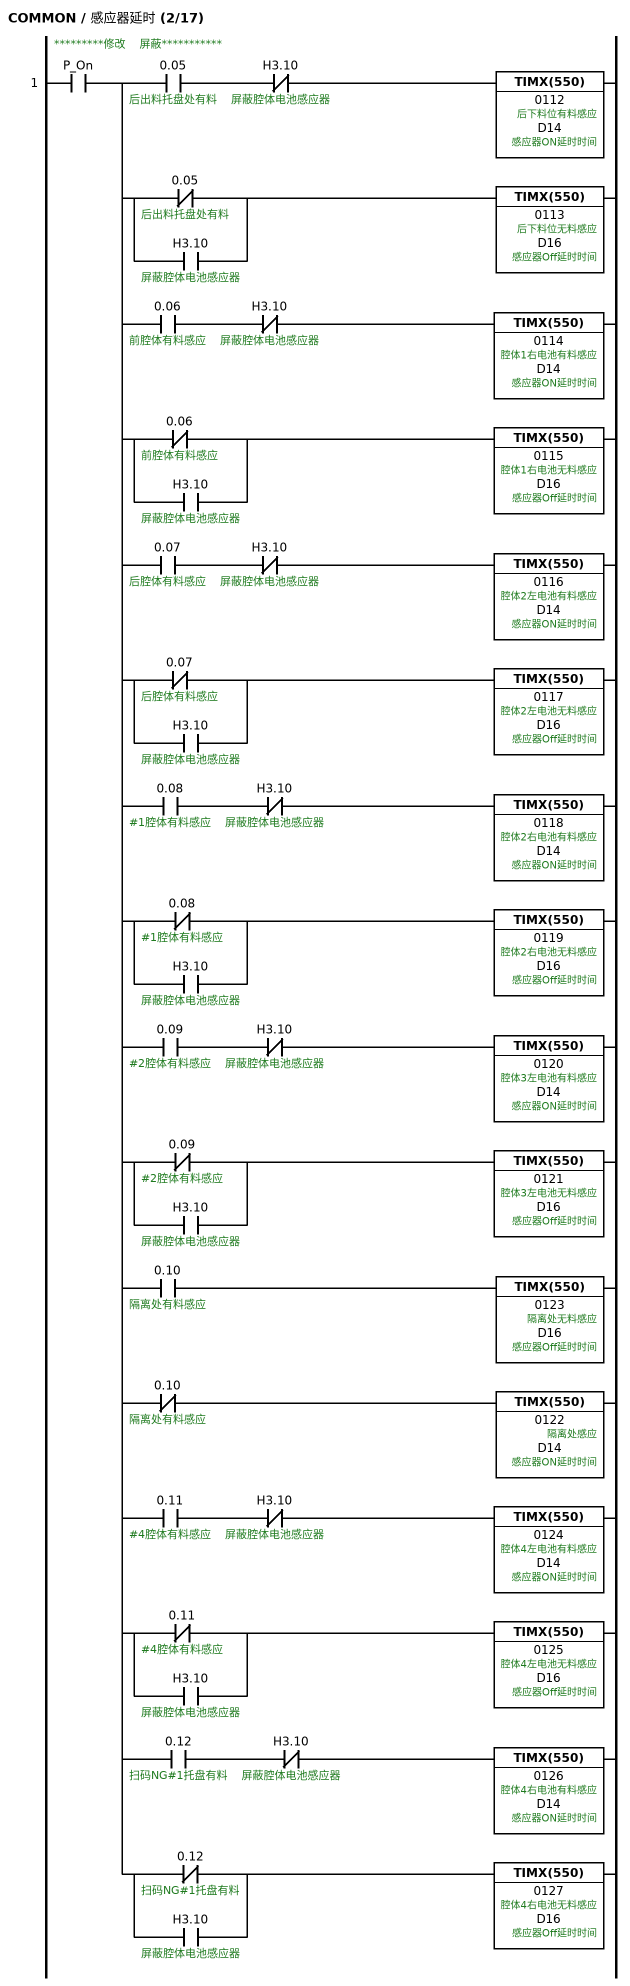
; [picture p408: COMMON / 感应器延时, rungs 1-1]
; rung 1: *********修改    屏蔽***********
LD P_On
OUT TR0
AND 0.05  ; 后出料托盘处有料
ANDNOT H3.10  ; 屏蔽腔体电池感应器
TIMX(550) 0112 D14  ; 感应器ON延时时间, 后下料位有料感应
LD TR0
LDNOT 0.05  ; 后出料托盘处有料
OR H3.10  ; 屏蔽腔体电池感应器
ANDLD
TIMX(550) 0113 D16  ; 感应器Off延时时间, 后下料位无料感应
LD TR0
AND 0.06  ; 前腔体有料感应
ANDNOT H3.10  ; 屏蔽腔体电池感应器
TIMX(550) 0114 D14  ; 感应器ON延时时间, 腔体1右电池有料感应
LD TR0
LDNOT 0.06  ; 前腔体有料感应
OR H3.10  ; 屏蔽腔体电池感应器
ANDLD
TIMX(550) 0115 D16  ; 感应器Off延时时间, 腔体1右电池无料感应
LD TR0
AND 0.07  ; 后腔体有料感应
ANDNOT H3.10  ; 屏蔽腔体电池感应器
TIMX(550) 0116 D14  ; 感应器ON延时时间, 腔体2左电池有料感应
LD TR0
LDNOT 0.07  ; 后腔体有料感应
OR H3.10  ; 屏蔽腔体电池感应器
ANDLD
TIMX(550) 0117 D16  ; 感应器Off延时时间, 腔体2左电池无料感应
LD TR0
AND 0.08  ; #1腔体有料感应
ANDNOT H3.10  ; 屏蔽腔体电池感应器
TIMX(550) 0118 D14  ; 感应器ON延时时间, 腔体2右电池有料感应
LD TR0
LDNOT 0.08  ; #1腔体有料感应
OR H3.10  ; 屏蔽腔体电池感应器
ANDLD
TIMX(550) 0119 D16  ; 感应器Off延时时间, 腔体2右电池无料感应
LD TR0
AND 0.09  ; #2腔体有料感应
ANDNOT H3.10  ; 屏蔽腔体电池感应器
TIMX(550) 0120 D14  ; 感应器ON延时时间, 腔体3左电池有料感应
LD TR0
LDNOT 0.09  ; #2腔体有料感应
OR H3.10  ; 屏蔽腔体电池感应器
ANDLD
TIMX(550) 0121 D16  ; 感应器Off延时时间, 腔体3左电池无料感应
LD TR0
AND 0.10  ; 隔离处有料感应
TIMX(550) 0123 D16  ; 感应器Off延时时间, 隔离处无料感应
LD TR0
ANDNOT 0.10  ; 隔离处有料感应
TIMX(550) 0122 D14  ; 感应器ON延时时间, 隔离处感应
LD TR0
AND 0.11  ; #4腔体有料感应
ANDNOT H3.10  ; 屏蔽腔体电池感应器
TIMX(550) 0124 D14  ; 感应器ON延时时间, 腔体4左电池有料感应
LD TR0
LDNOT 0.11  ; #4腔体有料感应
OR H3.10  ; 屏蔽腔体电池感应器
ANDLD
TIMX(550) 0125 D16  ; 感应器Off延时时间, 腔体4左电池无料感应
LD TR0
AND 0.12  ; 扫码NG#1托盘有料
ANDNOT H3.10  ; 屏蔽腔体电池感应器
TIMX(550) 0126 D14  ; 感应器ON延时时间, 腔体4右电池有料感应
LD TR0
LDNOT 0.12  ; 扫码NG#1托盘有料
OR H3.10  ; 屏蔽腔体电池感应器
ANDLD
TIMX(550) 0127 D16  ; 感应器Off延时时间, 腔体4右电池无料感应

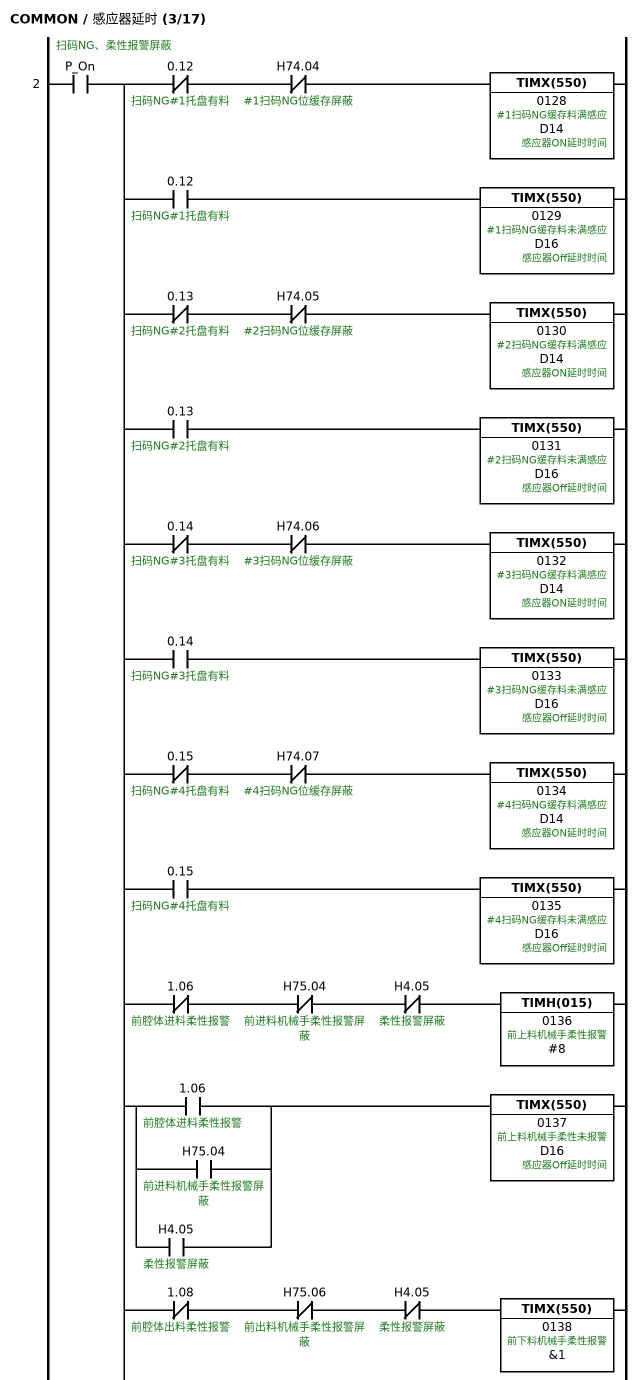

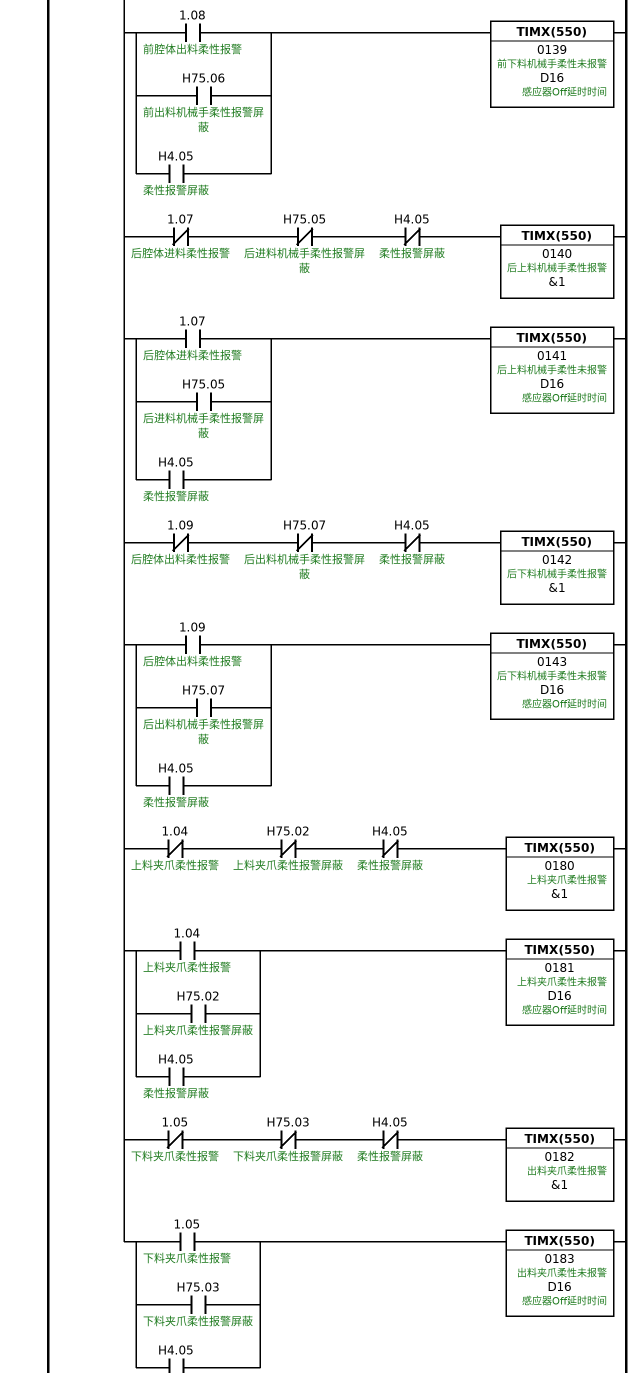

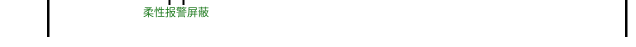
; rung 2: 扫码NG、柔性报警屏蔽
LD P_On
OUT TR0
ANDNOT 0.12  ; 扫码NG#1托盘有料
ANDNOT H74.04  ; #1扫码NG位缓存屏蔽
TIMX(550) 0128 D14  ; 感应器ON延时时间, #1扫码NG缓存料满感应
LD TR0
AND 0.12  ; 扫码NG#1托盘有料
TIMX(550) 0129 D16  ; 感应器Off延时时间, #1扫码NG缓存料未满感应
LD TR0
ANDNOT 0.13  ; 扫码NG#2托盘有料
ANDNOT H74.05  ; #2扫码NG位缓存屏蔽
TIMX(550) 0130 D14  ; 感应器ON延时时间, #2扫码NG缓存料满感应
LD TR0
AND 0.13  ; 扫码NG#2托盘有料
TIMX(550) 0131 D16  ; 感应器Off延时时间, #2扫码NG缓存料未满感应
LD TR0
ANDNOT 0.14  ; 扫码NG#3托盘有料
ANDNOT H74.06  ; #3扫码NG位缓存屏蔽
TIMX(550) 0132 D14  ; 感应器ON延时时间, #3扫码NG缓存料满感应
LD TR0
AND 0.14  ; 扫码NG#3托盘有料
TIMX(550) 0133 D16  ; 感应器Off延时时间, #3扫码NG缓存料未满感应
LD TR0
ANDNOT 0.15  ; 扫码NG#4托盘有料
ANDNOT H74.07  ; #4扫码NG位缓存屏蔽
TIMX(550) 0134 D14  ; 感应器ON延时时间, #4扫码NG缓存料满感应
LD TR0
AND 0.15  ; 扫码NG#4托盘有料
TIMX(550) 0135 D16  ; 感应器Off延时时间, #4扫码NG缓存料未满感应
LD TR0
ANDNOT 1.06  ; 前腔体进料柔性报警
ANDNOT H75.04  ; 前进料机械手柔性报警屏蔽
ANDNOT H4.05  ; 柔性报警屏蔽
TIMH(015) 0136 #8  ; 前上料机械手柔性报警
LD TR0
LD 1.06  ; 前腔体进料柔性报警
OR H75.04  ; 前进料机械手柔性报警屏蔽
OR H4.05  ; 柔性报警屏蔽
ANDLD
TIMX(550) 0137 D16  ; 感应器Off延时时间, 前上料机械手柔性未报警
LD TR0
ANDNOT 1.08  ; 前腔体出料柔性报警
ANDNOT H75.06  ; 前出料机械手柔性报警屏蔽
ANDNOT H4.05  ; 柔性报警屏蔽
TIMX(550) 0138 &1  ; 前下料机械手柔性报警
LD TR0
LD 1.08  ; 前腔体出料柔性报警
OR H75.06  ; 前出料机械手柔性报警屏蔽
OR H4.05  ; 柔性报警屏蔽
ANDLD
TIMX(550) 0139 D16  ; 感应器Off延时时间, 前下料机械手柔性未报警
LD TR0
ANDNOT 1.07  ; 后腔体进料柔性报警
ANDNOT H75.05  ; 后进料机械手柔性报警屏蔽
ANDNOT H4.05  ; 柔性报警屏蔽
TIMX(550) 0140 &1  ; 后上料机械手柔性报警
LD TR0
LD 1.07  ; 后腔体进料柔性报警
OR H75.05  ; 后进料机械手柔性报警屏蔽
OR H4.05  ; 柔性报警屏蔽
ANDLD
TIMX(550) 0141 D16  ; 感应器Off延时时间, 后上料机械手柔性未报警
LD TR0
ANDNOT 1.09  ; 后腔体出料柔性报警
ANDNOT H75.07  ; 后出料机械手柔性报警屏蔽
ANDNOT H4.05  ; 柔性报警屏蔽
TIMX(550) 0142 &1  ; 后下料机械手柔性报警
LD TR0
LD 1.09  ; 后腔体出料柔性报警
OR H75.07  ; 后出料机械手柔性报警屏蔽
OR H4.05  ; 柔性报警屏蔽
ANDLD
TIMX(550) 0143 D16  ; 感应器Off延时时间, 后下料机械手柔性未报警
LD TR0
ANDNOT 1.04  ; 上料夹爪柔性报警
ANDNOT H75.02  ; 上料夹爪柔性报警屏蔽
ANDNOT H4.05  ; 柔性报警屏蔽
TIMX(550) 0180 &1  ; 上料夹爪柔性报警
LD TR0
LD 1.04  ; 上料夹爪柔性报警
OR H75.02  ; 上料夹爪柔性报警屏蔽
OR H4.05  ; 柔性报警屏蔽
ANDLD
TIMX(550) 0181 D16  ; 感应器Off延时时间, 上料夹爪柔性未报警
LD TR0
ANDNOT 1.05  ; 下料夹爪柔性报警
ANDNOT H75.03  ; 下料夹爪柔性报警屏蔽
ANDNOT H4.05  ; 柔性报警屏蔽
TIMX(550) 0182 &1  ; 出料夹爪柔性报警
LD TR0
LD 1.05  ; 下料夹爪柔性报警
OR H75.03  ; 下料夹爪柔性报警屏蔽
OR H4.05  ; 柔性报警屏蔽
ANDLD
TIMX(550) 0183 D16  ; 感应器Off延时时间, 出料夹爪柔性未报警

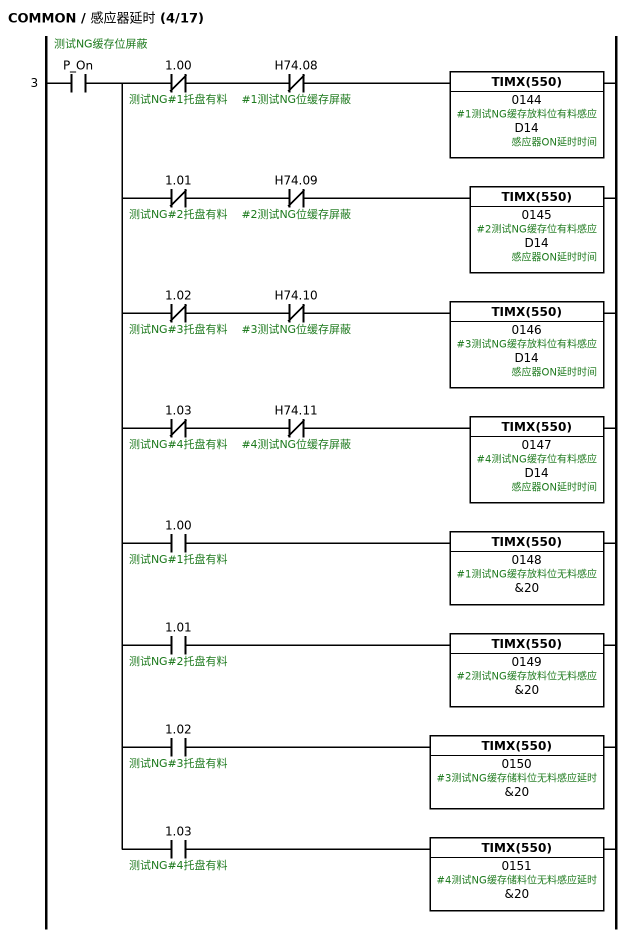
; rung 3: 测试NG缓存位屏蔽
LD P_On
OUT TR0
ANDNOT 1.00  ; 测试NG#1托盘有料
ANDNOT H74.08  ; #1测试NG位缓存屏蔽
TIMX(550) 0144 D14  ; 感应器ON延时时间, #1测试NG缓存放料位有料感应
LD TR0
ANDNOT 1.01  ; 测试NG#2托盘有料
ANDNOT H74.09  ; #2测试NG位缓存屏蔽
TIMX(550) 0145 D14  ; 感应器ON延时时间, #2测试NG缓存位有料感应
LD TR0
ANDNOT 1.02  ; 测试NG#3托盘有料
ANDNOT H74.10  ; #3测试NG位缓存屏蔽
TIMX(550) 0146 D14  ; 感应器ON延时时间, #3测试NG缓存放料位有料感应
LD TR0
ANDNOT 1.03  ; 测试NG#4托盘有料
ANDNOT H74.11  ; #4测试NG位缓存屏蔽
TIMX(550) 0147 D14  ; 感应器ON延时时间, #4测试NG缓存位有料感应
LD TR0
AND 1.00  ; 测试NG#1托盘有料
TIMX(550) 0148 &20  ; #1测试NG缓存放料位无料感应
LD TR0
AND 1.01  ; 测试NG#2托盘有料
TIMX(550) 0149 &20  ; #2测试NG缓存放料位无料感应
LD TR0
AND 1.02  ; 测试NG#3托盘有料
TIMX(550) 0150 &20  ; #3测试NG缓存储料位无料感应延时
LD TR0
AND 1.03  ; 测试NG#4托盘有料
TIMX(550) 0151 &20  ; #4测试NG缓存储料位无料感应延时

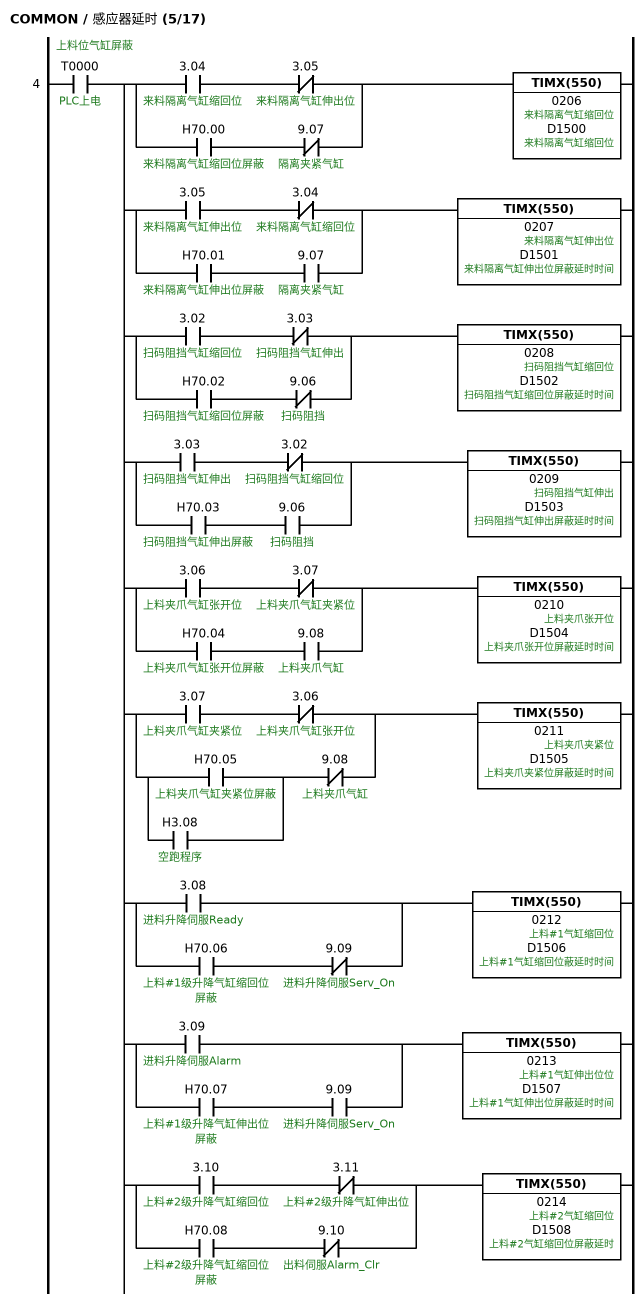

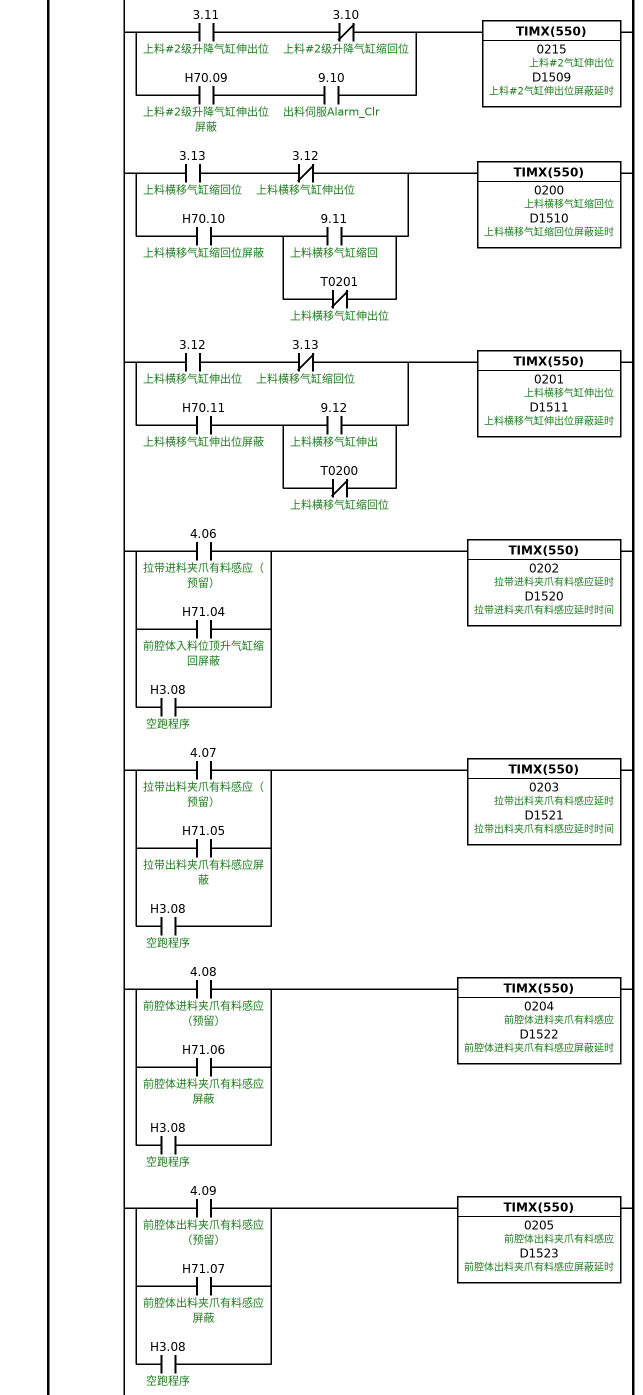

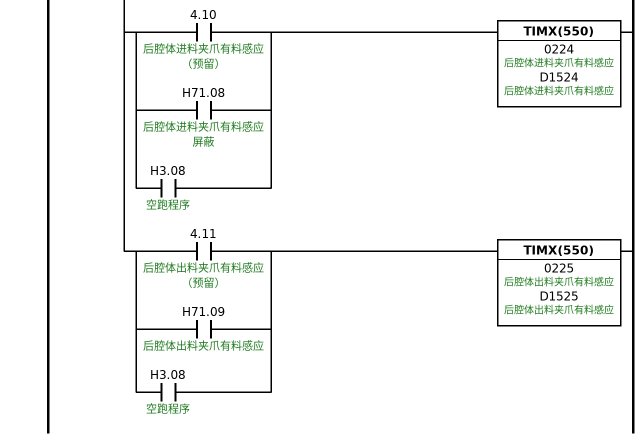
; rung 4: 上料位气缸屏蔽
LD T0000  ; PLC上电
OUT TR0
LD 3.04  ; 来料隔离气缸缩回位
ANDNOT 3.05  ; 来料隔离气缸伸出位
LD H70.00  ; 来料隔离气缸缩回位屏蔽
ANDNOT 9.07  ; 隔离夹紧气缸
ORLD
ANDLD
TIMX(550) 0206 D1500  ; 来料隔离气缸缩回位
LD TR0
LD 3.05  ; 来料隔离气缸伸出位
ANDNOT 3.04  ; 来料隔离气缸缩回位
LD H70.01  ; 来料隔离气缸伸出位屏蔽
AND 9.07  ; 隔离夹紧气缸
ORLD
ANDLD
TIMX(550) 0207 D1501  ; 来料隔离气缸伸出位屏蔽延时时间, 来料隔离气缸伸出位
LD TR0
LD 3.02  ; 扫码阻挡气缸缩回位
ANDNOT 3.03  ; 扫码阻挡气缸伸出
LD H70.02  ; 扫码阻挡气缸缩回位屏蔽
ANDNOT 9.06  ; 扫码阻挡
ORLD
ANDLD
TIMX(550) 0208 D1502  ; 扫码阻挡气缸缩回位屏蔽延时时间, 扫码阻挡气缸缩回位
LD TR0
LD 3.03  ; 扫码阻挡气缸伸出
ANDNOT 3.02  ; 扫码阻挡气缸缩回位
LD H70.03  ; 扫码阻挡气缸伸出屏蔽
AND 9.06  ; 扫码阻挡
ORLD
ANDLD
TIMX(550) 0209 D1503  ; 扫码阻挡气缸伸出屏蔽延时时间, 扫码阻挡气缸伸出
LD TR0
LD 3.06  ; 上料夹爪气缸张开位
ANDNOT 3.07  ; 上料夹爪气缸夹紧位
LD H70.04  ; 上料夹爪气缸张开位屏蔽
AND 9.08  ; 上料夹爪气缸
ORLD
ANDLD
TIMX(550) 0210 D1504  ; 上料夹爪张开位屏蔽延时时间, 上料夹爪张开位
LD TR0
LD 3.07  ; 上料夹爪气缸夹紧位
ANDNOT 3.06  ; 上料夹爪气缸张开位
LD H70.05  ; 上料夹爪气缸夹紧位屏蔽
OR H3.08  ; 空跑程序
ANDNOT 9.08  ; 上料夹爪气缸
ORLD
ANDLD
TIMX(550) 0211 D1505  ; 上料夹爪夹紧位屏蔽延时时间, 上料夹爪夹紧位
LD TR0
LD 3.08  ; 进料升降伺服Ready
LD H70.06  ; 上料#1级升降气缸缩回位屏蔽
ANDNOT 9.09  ; 进料升降伺服Serv_On
ORLD
ANDLD
TIMX(550) 0212 D1506  ; 上料#1气缸缩回位蔽延时时间, 上料#1气缸缩回位
LD TR0
LD 3.09  ; 进料升降伺服Alarm
LD H70.07  ; 上料#1级升降气缸伸出位屏蔽
AND 9.09  ; 进料升降伺服Serv_On
ORLD
ANDLD
TIMX(550) 0213 D1507  ; 上料#1气缸伸出位屏蔽延时时间, 上料#1气缸伸出位位
LD TR0
LD 3.10  ; 上料#2级升降气缸缩回位
ANDNOT 3.11  ; 上料#2级升降气缸伸出位
LD H70.08  ; 上料#2级升降气缸缩回位屏蔽
ANDNOT 9.10  ; 出料伺服Alarm_Clr
ORLD
ANDLD
TIMX(550) 0214 D1508  ; 上料#2气缸缩回位屏蔽延时, 上料#2气缸缩回位
LD TR0
LD 3.11  ; 上料#2级升降气缸伸出位
ANDNOT 3.10  ; 上料#2级升降气缸缩回位
LD H70.09  ; 上料#2级升降气缸伸出位屏蔽
AND 9.10  ; 出料伺服Alarm_Clr
ORLD
ANDLD
TIMX(550) 0215 D1509  ; 上料#2气缸伸出位屏蔽延时, 上料#2气缸伸出位
LD TR0
LD 3.13  ; 上料横移气缸缩回位
ANDNOT 3.12  ; 上料横移气缸伸出位
LD H70.10  ; 上料横移气缸缩回位屏蔽
LD 9.11  ; 上料横移气缸缩回
ORNOT T0201  ; 上料横移气缸伸出位
ANDLD
ORLD
ANDLD
TIMX(550) 0200 D1510  ; 上料横移气缸缩回位屏蔽延时, 上料横移气缸缩回位
LD TR0
LD 3.12  ; 上料横移气缸伸出位
ANDNOT 3.13  ; 上料横移气缸缩回位
LD H70.11  ; 上料横移气缸伸出位屏蔽
LD 9.12  ; 上料横移气缸伸出
ORNOT T0200  ; 上料横移气缸缩回位
ANDLD
ORLD
ANDLD
TIMX(550) 0201 D1511  ; 上料横移气缸伸出位屏蔽延时, 上料横移气缸伸出位
LD TR0
LD 4.06  ; 拉带进料夹爪有料感应（预留）
OR H71.04  ; 前腔体入料位顶升气缸缩回屏蔽
OR H3.08  ; 空跑程序
ANDLD
TIMX(550) 0202 D1520  ; 拉带进料夹爪有料感应延时时间, 拉带进料夹爪有料感应延时
LD TR0
LD 4.07  ; 拉带出料夹爪有料感应（预留）
OR H71.05  ; 拉带出料夹爪有料感应屏蔽
OR H3.08  ; 空跑程序
ANDLD
TIMX(550) 0203 D1521  ; 拉带出料夹爪有料感应延时时间, 拉带出料夹爪有料感应延时
LD TR0
LD 4.08  ; 前腔体进料夹爪有料感应（预留）
OR H71.06  ; 前腔体进料夹爪有料感应屏蔽
OR H3.08  ; 空跑程序
ANDLD
TIMX(550) 0204 D1522  ; 前腔体进料夹爪有料感应屏蔽延时, 前腔体进料夹爪有料感应
LD TR0
LD 4.09  ; 前腔体出料夹爪有料感应（预留）
OR H71.07  ; 前腔体出料夹爪有料感应屏蔽
OR H3.08  ; 空跑程序
ANDLD
TIMX(550) 0205 D1523  ; 前腔体出料夹爪有料感应屏蔽延时, 前腔体出料夹爪有料感应
LD TR0
LD 4.10  ; 后腔体进料夹爪有料感应（预留）
OR H71.08  ; 后腔体进料夹爪有料感应屏蔽
OR H3.08  ; 空跑程序
ANDLD
TIMX(550) 0224 D1524  ; 后腔体进料夹爪有料感应
LD TR0
LD 4.11  ; 后腔体出料夹爪有料感应（预留）
OR H71.09  ; 后腔体出料夹爪有料感应
OR H3.08  ; 空跑程序
ANDLD
TIMX(550) 0225 D1525  ; 后腔体出料夹爪有料感应

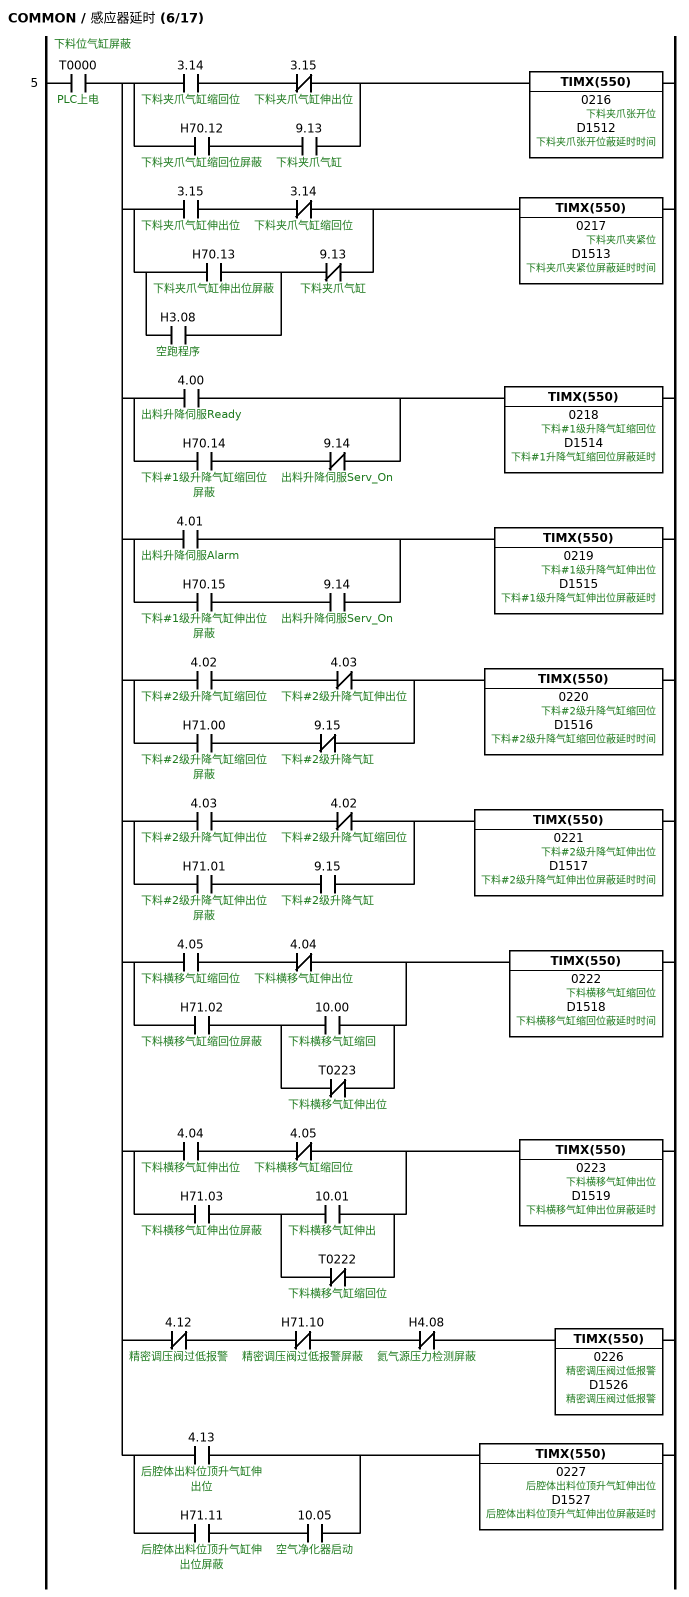
; rung 5: 下料位气缸屏蔽
LD T0000  ; PLC上电
OUT TR0
LD 3.14  ; 下料夹爪气缸缩回位
ANDNOT 3.15  ; 下料夹爪气缸伸出位
LD H70.12  ; 下料夹爪气缸缩回位屏蔽
AND 9.13  ; 下料夹爪气缸
ORLD
ANDLD
TIMX(550) 0216 D1512  ; 下料夹爪张开位蔽延时时间, 下料夹爪张开位
LD TR0
LD 3.15  ; 下料夹爪气缸伸出位
ANDNOT 3.14  ; 下料夹爪气缸缩回位
LD H70.13  ; 下料夹爪气缸伸出位屏蔽
OR H3.08  ; 空跑程序
ANDNOT 9.13  ; 下料夹爪气缸
ORLD
ANDLD
TIMX(550) 0217 D1513  ; 下料夹爪夹紧位屏蔽延时时间, 下料夹爪夹紧位
LD TR0
LD 4.00  ; 出料升降伺服Ready
LD H70.14  ; 下料#1级升降气缸缩回位屏蔽
ANDNOT 9.14  ; 出料升降伺服Serv_On
ORLD
ANDLD
TIMX(550) 0218 D1514  ; 下料#1升降气缸缩回位屏蔽延时, 下料#1级升降气缸缩回位
LD TR0
LD 4.01  ; 出料升降伺服Alarm
LD H70.15  ; 下料#1级升降气缸伸出位屏蔽
AND 9.14  ; 出料升降伺服Serv_On
ORLD
ANDLD
TIMX(550) 0219 D1515  ; 下料#1级升降气缸伸出位屏蔽延时, 下料#1级升降气缸伸出位
LD TR0
LD 4.02  ; 下料#2级升降气缸缩回位
ANDNOT 4.03  ; 下料#2级升降气缸伸出位
LD H71.00  ; 下料#2级升降气缸缩回位屏蔽
ANDNOT 9.15  ; 下料#2级升降气缸
ORLD
ANDLD
TIMX(550) 0220 D1516  ; 下料#2级升降气缸缩回位蔽延时时间, 下料#2级升降气缸缩回位
LD TR0
LD 4.03  ; 下料#2级升降气缸伸出位
ANDNOT 4.02  ; 下料#2级升降气缸缩回位
LD H71.01  ; 下料#2级升降气缸伸出位屏蔽
AND 9.15  ; 下料#2级升降气缸
ORLD
ANDLD
TIMX(550) 0221 D1517  ; 下料#2级升降气缸伸出位屏蔽延时时间, 下料#2级升降气缸伸出位
LD TR0
LD 4.05  ; 下料横移气缸缩回位
ANDNOT 4.04  ; 下料横移气缸伸出位
LD H71.02  ; 下料横移气缸缩回位屏蔽
LD 10.00  ; 下料横移气缸缩回
ORNOT T0223  ; 下料横移气缸伸出位
ANDLD
ORLD
ANDLD
TIMX(550) 0222 D1518  ; 下料横移气缸缩回位蔽延时时间, 下料横移气缸缩回位
LD TR0
LD 4.04  ; 下料横移气缸伸出位
ANDNOT 4.05  ; 下料横移气缸缩回位
LD H71.03  ; 下料横移气缸伸出位屏蔽
LD 10.01  ; 下料横移气缸伸出
ORNOT T0222  ; 下料横移气缸缩回位
ANDLD
ORLD
ANDLD
TIMX(550) 0223 D1519  ; 下料横移气缸伸出位屏蔽延时, 下料横移气缸伸出位
LD TR0
ANDNOT 4.12  ; 精密调压阀过低报警
ANDNOT H71.10  ; 精密调压阀过低报警屏蔽
ANDNOT H4.08  ; 氦气源压力检测屏蔽
TIMX(550) 0226 D1526  ; 精密调压阀过低报警
LD TR0
LD 4.13  ; 后腔体出料位顶升气缸伸出位
LD H71.11  ; 后腔体出料位顶升气缸伸出位屏蔽
AND 10.05  ; 空气净化器启动
ORLD
ANDLD
TIMX(550) 0227 D1527  ; 后腔体出料位顶升气缸伸出位屏蔽延时, 后腔体出料位顶升气缸伸出位

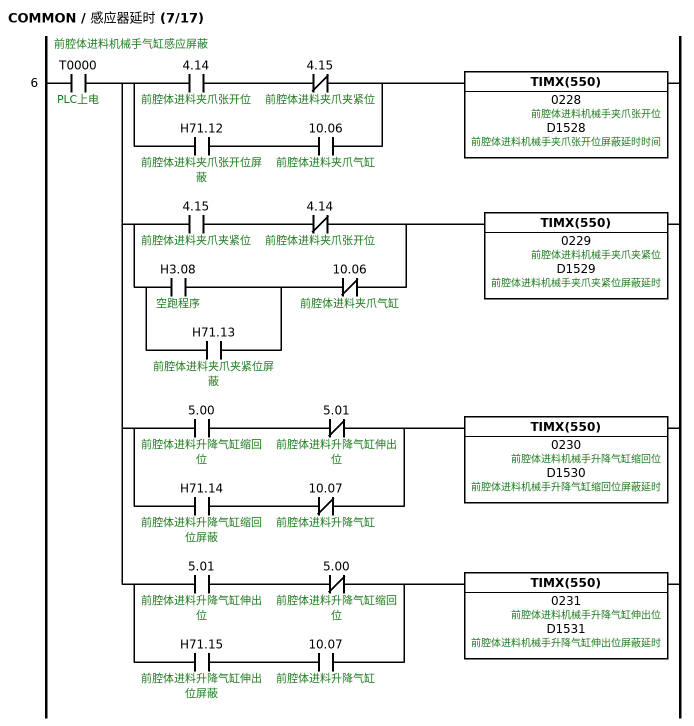
; rung 6: 前腔体进料机械手气缸感应屏蔽
LD T0000  ; PLC上电
OUT TR0
LD 4.14  ; 前腔体进料夹爪张开位
ANDNOT 4.15  ; 前腔体进料夹爪夹紧位
LD H71.12  ; 前腔体进料夹爪张开位屏蔽
AND 10.06  ; 前腔体进料夹爪气缸
ORLD
ANDLD
TIMX(550) 0228 D1528  ; 前腔体进料机械手夹爪张开位屏蔽延时时间, 前腔体进料机械手夹爪张开位
LD TR0
LD 4.15  ; 前腔体进料夹爪夹紧位
ANDNOT 4.14  ; 前腔体进料夹爪张开位
LD H3.08  ; 空跑程序
OR H71.13  ; 前腔体进料夹爪夹紧位屏蔽
ANDNOT 10.06  ; 前腔体进料夹爪气缸
ORLD
ANDLD
TIMX(550) 0229 D1529  ; 前腔体进料机械手夹爪夹紧位屏蔽延时, 前腔体进料机械手夹爪夹紧位
LD TR0
LD 5.00  ; 前腔体进料升降气缸缩回位
ANDNOT 5.01  ; 前腔体进料升降气缸伸出位
LD H71.14  ; 前腔体进料升降气缸缩回位屏蔽
ANDNOT 10.07  ; 前腔体进料升降气缸
ORLD
ANDLD
TIMX(550) 0230 D1530  ; 前腔体进料机械手升降气缸缩回位屏蔽延时, 前腔体进料机械手升降气缸缩回位
LD TR0
LD 5.01  ; 前腔体进料升降气缸伸出位
ANDNOT 5.00  ; 前腔体进料升降气缸缩回位
LD H71.15  ; 前腔体进料升降气缸伸出位屏蔽
AND 10.07  ; 前腔体进料升降气缸
ORLD
ANDLD
TIMX(550) 0231 D1531  ; 前腔体进料机械手升降气缸伸出位屏蔽延时, 前腔体进料机械手升降气缸伸出位

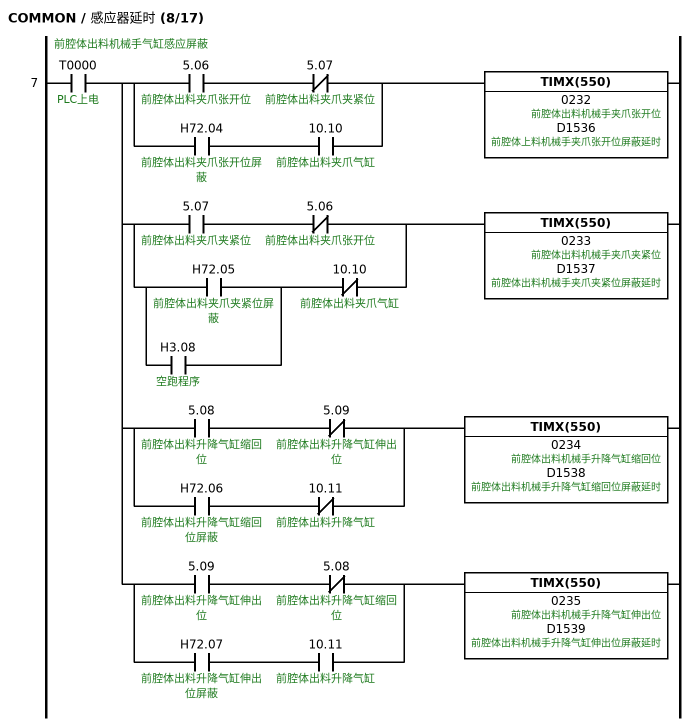
; rung 7: 前腔体出料机械手气缸感应屏蔽
LD T0000  ; PLC上电
OUT TR0
LD 5.06  ; 前腔体出料夹爪张开位
ANDNOT 5.07  ; 前腔体出料夹爪夹紧位
LD H72.04  ; 前腔体出料夹爪张开位屏蔽
AND 10.10  ; 前腔体出料夹爪气缸
ORLD
ANDLD
TIMX(550) 0232 D1536  ; 前腔体上料机械手夹爪张开位屏蔽延时, 前腔体出料机械手夹爪张开位
LD TR0
LD 5.07  ; 前腔体出料夹爪夹紧位
ANDNOT 5.06  ; 前腔体出料夹爪张开位
LD H72.05  ; 前腔体出料夹爪夹紧位屏蔽
OR H3.08  ; 空跑程序
ANDNOT 10.10  ; 前腔体出料夹爪气缸
ORLD
ANDLD
TIMX(550) 0233 D1537  ; 前腔体出料机械手夹爪夹紧位屏蔽延时, 前腔体出料机械手夹爪夹紧位
LD TR0
LD 5.08  ; 前腔体出料升降气缸缩回位
ANDNOT 5.09  ; 前腔体出料升降气缸伸出位
LD H72.06  ; 前腔体出料升降气缸缩回位屏蔽
ANDNOT 10.11  ; 前腔体出料升降气缸
ORLD
ANDLD
TIMX(550) 0234 D1538  ; 前腔体出料机械手升降气缸缩回位屏蔽延时, 前腔体出料机械手升降气缸缩回位
LD TR0
LD 5.09  ; 前腔体出料升降气缸伸出位
ANDNOT 5.08  ; 前腔体出料升降气缸缩回位
LD H72.07  ; 前腔体出料升降气缸伸出位屏蔽
AND 10.11  ; 前腔体出料升降气缸
ORLD
ANDLD
TIMX(550) 0235 D1539  ; 前腔体出料机械手升降气缸伸出位屏蔽延时, 前腔体出料机械手升降气缸伸出位

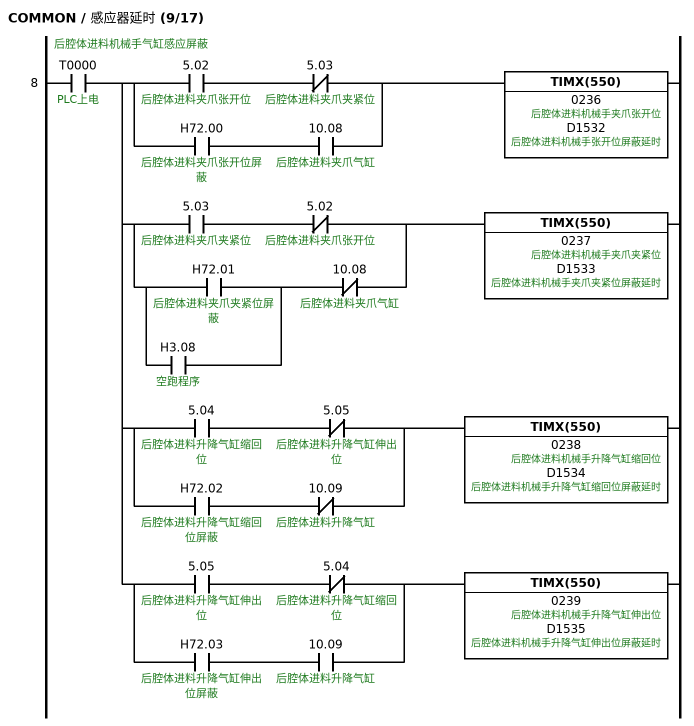
; rung 8: 后腔体进料机械手气缸感应屏蔽
LD T0000  ; PLC上电
OUT TR0
LD 5.02  ; 后腔体进料夹爪张开位
ANDNOT 5.03  ; 后腔体进料夹爪夹紧位
LD H72.00  ; 后腔体进料夹爪张开位屏蔽
AND 10.08  ; 后腔体进料夹爪气缸
ORLD
ANDLD
TIMX(550) 0236 D1532  ; 后腔体进料机械手张开位屏蔽延时, 后腔体进料机械手夹爪张开位
LD TR0
LD 5.03  ; 后腔体进料夹爪夹紧位
ANDNOT 5.02  ; 后腔体进料夹爪张开位
LD H72.01  ; 后腔体进料夹爪夹紧位屏蔽
OR H3.08  ; 空跑程序
ANDNOT 10.08  ; 后腔体进料夹爪气缸
ORLD
ANDLD
TIMX(550) 0237 D1533  ; 后腔体进料机械手夹爪夹紧位屏蔽延时, 后腔体进料机械手夹爪夹紧位
LD TR0
LD 5.04  ; 后腔体进料升降气缸缩回位
ANDNOT 5.05  ; 后腔体进料升降气缸伸出位
LD H72.02  ; 后腔体进料升降气缸缩回位屏蔽
ANDNOT 10.09  ; 后腔体进料升降气缸
ORLD
ANDLD
TIMX(550) 0238 D1534  ; 后腔体进料机械手升降气缸缩回位屏蔽延时, 后腔体进料机械手升降气缸缩回位
LD TR0
LD 5.05  ; 后腔体进料升降气缸伸出位
ANDNOT 5.04  ; 后腔体进料升降气缸缩回位
LD H72.03  ; 后腔体进料升降气缸伸出位屏蔽
AND 10.09  ; 后腔体进料升降气缸
ORLD
ANDLD
TIMX(550) 0239 D1535  ; 后腔体进料机械手升降气缸伸出位屏蔽延时, 后腔体进料机械手升降气缸伸出位

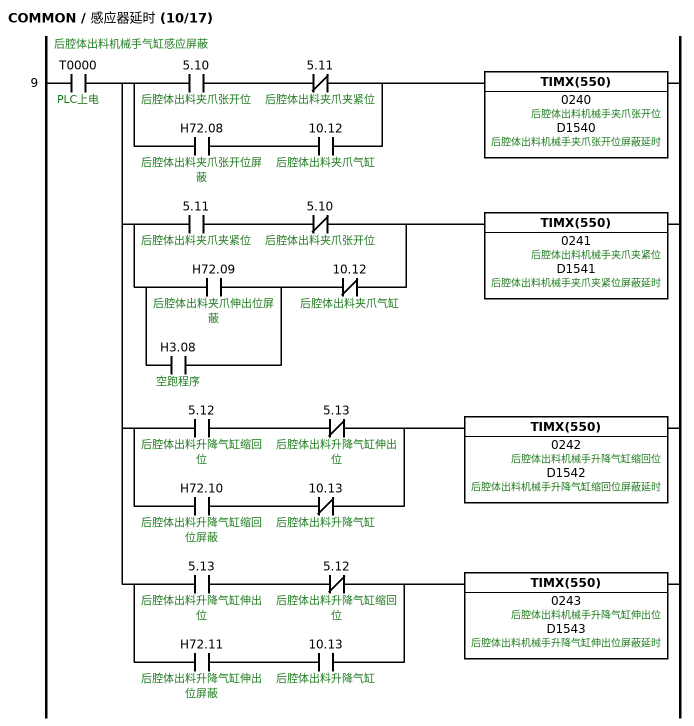
; rung 9: 后腔体出料机械手气缸感应屏蔽
LD T0000  ; PLC上电
OUT TR0
LD 5.10  ; 后腔体出料夹爪张开位
ANDNOT 5.11  ; 后腔体出料夹爪夹紧位
LD H72.08  ; 后腔体出料夹爪张开位屏蔽
AND 10.12  ; 后腔体出料夹爪气缸
ORLD
ANDLD
TIMX(550) 0240 D1540  ; 后腔体出料机械手夹爪张开位屏蔽延时, 后腔体出料机械手夹爪张开位
LD TR0
LD 5.11  ; 后腔体出料夹爪夹紧位
ANDNOT 5.10  ; 后腔体出料夹爪张开位
LD H72.09  ; 后腔体出料夹爪伸出位屏蔽
OR H3.08  ; 空跑程序
ANDNOT 10.12  ; 后腔体出料夹爪气缸
ORLD
ANDLD
TIMX(550) 0241 D1541  ; 后腔体出料机械手夹爪夹紧位屏蔽延时, 后腔体出料机械手夹爪夹紧位
LD TR0
LD 5.12  ; 后腔体出料升降气缸缩回位
ANDNOT 5.13  ; 后腔体出料升降气缸伸出位
LD H72.10  ; 后腔体出料升降气缸缩回位屏蔽
ANDNOT 10.13  ; 后腔体出料升降气缸
ORLD
ANDLD
TIMX(550) 0242 D1542  ; 后腔体出料机械手升降气缸缩回位屏蔽延时, 后腔体出料机械手升降气缸缩回位
LD TR0
LD 5.13  ; 后腔体出料升降气缸伸出位
ANDNOT 5.12  ; 后腔体出料升降气缸缩回位
LD H72.11  ; 后腔体出料升降气缸伸出位屏蔽
AND 10.13  ; 后腔体出料升降气缸
ORLD
ANDLD
TIMX(550) 0243 D1543  ; 后腔体出料机械手升降气缸伸出位屏蔽延时, 后腔体出料机械手升降气缸伸出位

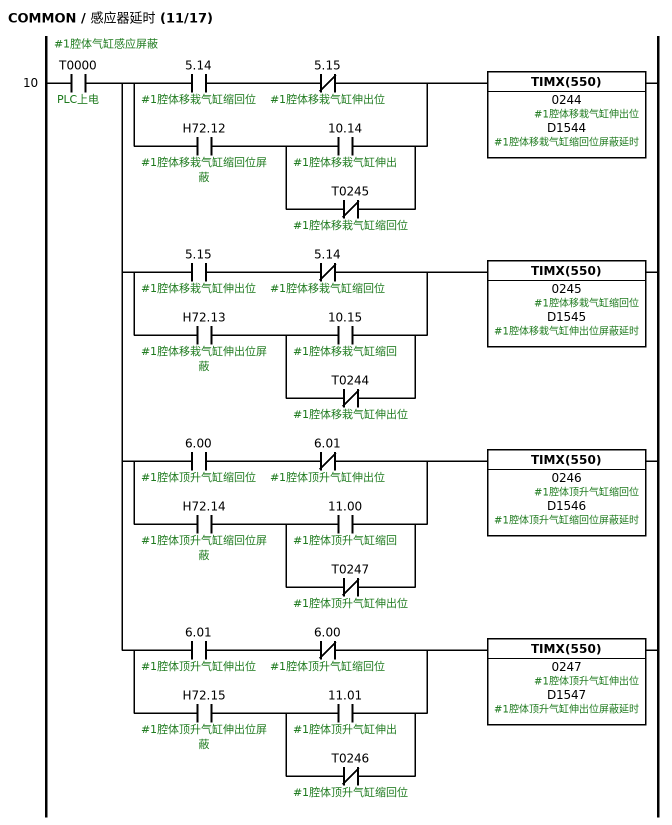
; rung 10: #1腔体气缸感应屏蔽
LD T0000  ; PLC上电
OUT TR0
LD 5.14  ; #1腔体移栽气缸缩回位
ANDNOT 5.15  ; #1腔体移栽气缸伸出位
LD H72.12  ; #1腔体移栽气缸缩回位屏蔽
LD 10.14  ; #1腔体移栽气缸伸出
ORNOT T0245  ; #1腔体移栽气缸缩回位
ANDLD
ORLD
ANDLD
TIMX(550) 0244 D1544  ; #1腔体移栽气缸缩回位屏蔽延时, #1腔体移栽气缸伸出位
LD TR0
LD 5.15  ; #1腔体移栽气缸伸出位
ANDNOT 5.14  ; #1腔体移栽气缸缩回位
LD H72.13  ; #1腔体移栽气缸伸出位屏蔽
LD 10.15  ; #1腔体移栽气缸缩回
ORNOT T0244  ; #1腔体移栽气缸伸出位
ANDLD
ORLD
ANDLD
TIMX(550) 0245 D1545  ; #1腔体移栽气缸伸出位屏蔽延时, #1腔体移栽气缸缩回位
LD TR0
LD 6.00  ; #1腔体顶升气缸缩回位
ANDNOT 6.01  ; #1腔体顶升气缸伸出位
LD H72.14  ; #1腔体顶升气缸缩回位屏蔽
LD 11.00  ; #1腔体顶升气缸缩回
ORNOT T0247  ; #1腔体顶升气缸伸出位
ANDLD
ORLD
ANDLD
TIMX(550) 0246 D1546  ; #1腔体顶升气缸缩回位屏蔽延时, #1腔体顶升气缸缩回位
LD TR0
LD 6.01  ; #1腔体顶升气缸伸出位
ANDNOT 6.00  ; #1腔体顶升气缸缩回位
LD H72.15  ; #1腔体顶升气缸伸出位屏蔽
LD 11.01  ; #1腔体顶升气缸伸出
ORNOT T0246  ; #1腔体顶升气缸缩回位
ANDLD
ORLD
ANDLD
TIMX(550) 0247 D1547  ; #1腔体顶升气缸伸出位屏蔽延时, #1腔体顶升气缸伸出位

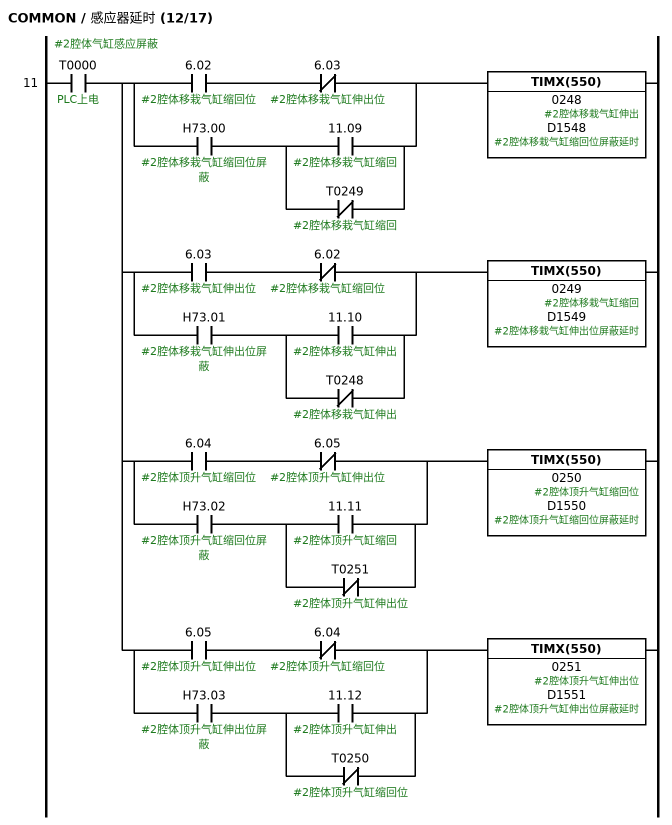
; rung 11: #2腔体气缸感应屏蔽
LD T0000  ; PLC上电
OUT TR0
LD 6.02  ; #2腔体移栽气缸缩回位
ANDNOT 6.03  ; #2腔体移栽气缸伸出位
LD H73.00  ; #2腔体移栽气缸缩回位屏蔽
LD 11.09  ; #2腔体移栽气缸缩回
ORNOT T0249  ; #2腔体移栽气缸缩回
ANDLD
ORLD
ANDLD
TIMX(550) 0248 D1548  ; #2腔体移栽气缸缩回位屏蔽延时, #2腔体移栽气缸伸出
LD TR0
LD 6.03  ; #2腔体移栽气缸伸出位
ANDNOT 6.02  ; #2腔体移栽气缸缩回位
LD H73.01  ; #2腔体移栽气缸伸出位屏蔽
LD 11.10  ; #2腔体移栽气缸伸出
ORNOT T0248  ; #2腔体移栽气缸伸出
ANDLD
ORLD
ANDLD
TIMX(550) 0249 D1549  ; #2腔体移栽气缸伸出位屏蔽延时, #2腔体移栽气缸缩回
LD TR0
LD 6.04  ; #2腔体顶升气缸缩回位
ANDNOT 6.05  ; #2腔体顶升气缸伸出位
LD H73.02  ; #2腔体顶升气缸缩回位屏蔽
LD 11.11  ; #2腔体顶升气缸缩回
ORNOT T0251  ; #2腔体顶升气缸伸出位
ANDLD
ORLD
ANDLD
TIMX(550) 0250 D1550  ; #2腔体顶升气缸缩回位屏蔽延时, #2腔体顶升气缸缩回位
LD TR0
LD 6.05  ; #2腔体顶升气缸伸出位
ANDNOT 6.04  ; #2腔体顶升气缸缩回位
LD H73.03  ; #2腔体顶升气缸伸出位屏蔽
LD 11.12  ; #2腔体顶升气缸伸出
ORNOT T0250  ; #2腔体顶升气缸缩回位
ANDLD
ORLD
ANDLD
TIMX(550) 0251 D1551  ; #2腔体顶升气缸伸出位屏蔽延时, #2腔体顶升气缸伸出位

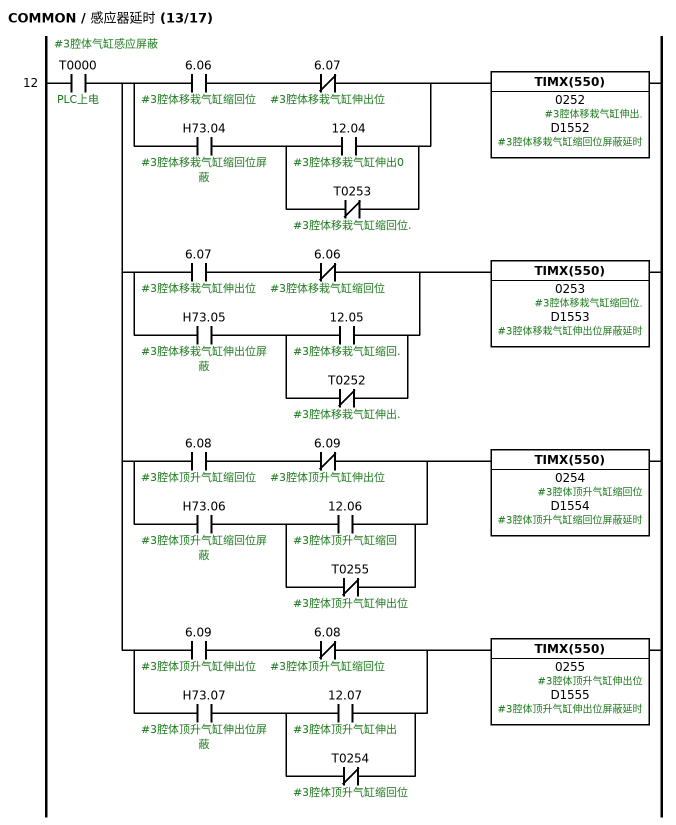
; rung 12: #3腔体气缸感应屏蔽
LD T0000  ; PLC上电
OUT TR0
LD 6.06  ; #3腔体移栽气缸缩回位
ANDNOT 6.07  ; #3腔体移栽气缸伸出位
LD H73.04  ; #3腔体移栽气缸缩回位屏蔽
LD 12.04  ; #3腔体移栽气缸伸出0
ORNOT T0253  ; #3腔体移栽气缸缩回位.
ANDLD
ORLD
ANDLD
TIMX(550) 0252 D1552  ; #3腔体移栽气缸缩回位屏蔽延时, #3腔体移栽气缸伸出.
LD TR0
LD 6.07  ; #3腔体移栽气缸伸出位
ANDNOT 6.06  ; #3腔体移栽气缸缩回位
LD H73.05  ; #3腔体移栽气缸伸出位屏蔽
LD 12.05  ; #3腔体移栽气缸缩回.
ORNOT T0252  ; #3腔体移栽气缸伸出.
ANDLD
ORLD
ANDLD
TIMX(550) 0253 D1553  ; #3腔体移栽气缸伸出位屏蔽延时, #3腔体移栽气缸缩回位.
LD TR0
LD 6.08  ; #3腔体顶升气缸缩回位
ANDNOT 6.09  ; #3腔体顶升气缸伸出位
LD H73.06  ; #3腔体顶升气缸缩回位屏蔽
LD 12.06  ; #3腔体顶升气缸缩回
ORNOT T0255  ; #3腔体顶升气缸伸出位
ANDLD
ORLD
ANDLD
TIMX(550) 0254 D1554  ; #3腔体顶升气缸缩回位屏蔽延时, #3腔体顶升气缸缩回位
LD TR0
LD 6.09  ; #3腔体顶升气缸伸出位
ANDNOT 6.08  ; #3腔体顶升气缸缩回位
LD H73.07  ; #3腔体顶升气缸伸出位屏蔽
LD 12.07  ; #3腔体顶升气缸伸出
ORNOT T0254  ; #3腔体顶升气缸缩回位
ANDLD
ORLD
ANDLD
TIMX(550) 0255 D1555  ; #3腔体顶升气缸伸出位屏蔽延时, #3腔体顶升气缸伸出位

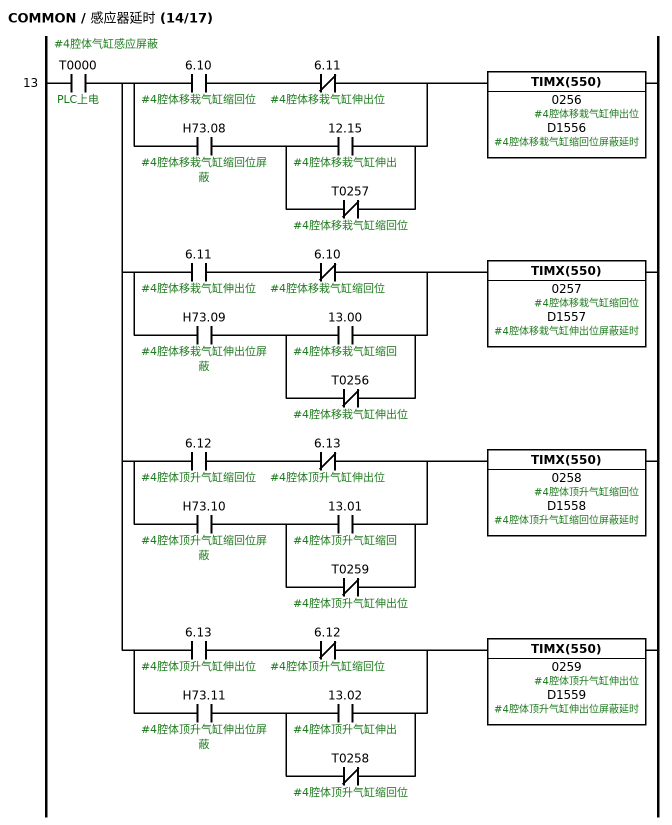
; rung 13: #4腔体气缸感应屏蔽
LD T0000  ; PLC上电
OUT TR0
LD 6.10  ; #4腔体移栽气缸缩回位
ANDNOT 6.11  ; #4腔体移栽气缸伸出位
LD H73.08  ; #4腔体移栽气缸缩回位屏蔽
LD 12.15  ; #4腔体移栽气缸伸出
ORNOT T0257  ; #4腔体移栽气缸缩回位
ANDLD
ORLD
ANDLD
TIMX(550) 0256 D1556  ; #4腔体移栽气缸缩回位屏蔽延时, #4腔体移栽气缸伸出位
LD TR0
LD 6.11  ; #4腔体移栽气缸伸出位
ANDNOT 6.10  ; #4腔体移栽气缸缩回位
LD H73.09  ; #4腔体移栽气缸伸出位屏蔽
LD 13.00  ; #4腔体移栽气缸缩回
ORNOT T0256  ; #4腔体移栽气缸伸出位
ANDLD
ORLD
ANDLD
TIMX(550) 0257 D1557  ; #4腔体移栽气缸伸出位屏蔽延时, #4腔体移栽气缸缩回位
LD TR0
LD 6.12  ; #4腔体顶升气缸缩回位
ANDNOT 6.13  ; #4腔体顶升气缸伸出位
LD H73.10  ; #4腔体顶升气缸缩回位屏蔽
LD 13.01  ; #4腔体顶升气缸缩回
ORNOT T0259  ; #4腔体顶升气缸伸出位
ANDLD
ORLD
ANDLD
TIMX(550) 0258 D1558  ; #4腔体顶升气缸缩回位屏蔽延时, #4腔体顶升气缸缩回位
LD TR0
LD 6.13  ; #4腔体顶升气缸伸出位
ANDNOT 6.12  ; #4腔体顶升气缸缩回位
LD H73.11  ; #4腔体顶升气缸伸出位屏蔽
LD 13.02  ; #4腔体顶升气缸伸出
ORNOT T0258  ; #4腔体顶升气缸缩回位
ANDLD
ORLD
ANDLD
TIMX(550) 0259 D1559  ; #4腔体顶升气缸伸出位屏蔽延时, #4腔体顶升气缸伸出位

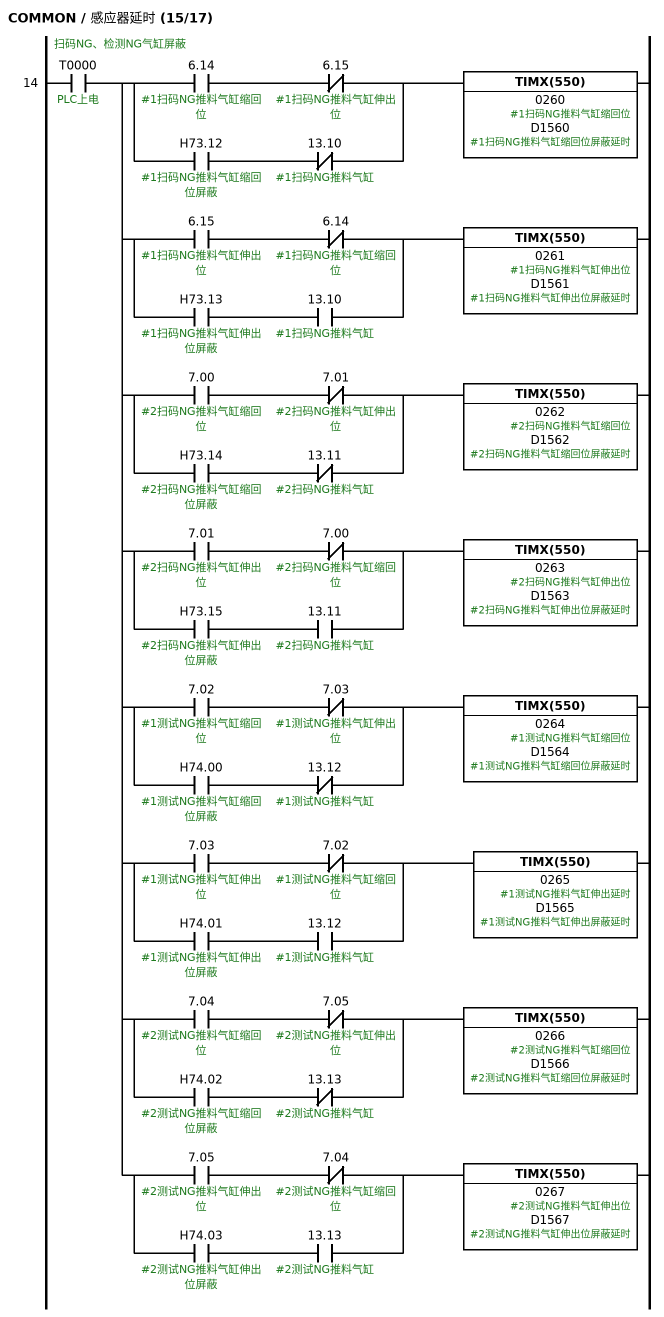
; rung 14: 扫码NG、检测NG气缸屏蔽
LD T0000  ; PLC上电
OUT TR0
LD 6.14  ; #1扫码NG推料气缸缩回位
ANDNOT 6.15  ; #1扫码NG推料气缸伸出位
LD H73.12  ; #1扫码NG推料气缸缩回位屏蔽
ANDNOT 13.10  ; #1扫码NG推料气缸
ORLD
ANDLD
TIMX(550) 0260 D1560  ; #1扫码NG推料气缸缩回位屏蔽延时, #1扫码NG推料气缸缩回位
LD TR0
LD 6.15  ; #1扫码NG推料气缸伸出位
ANDNOT 6.14  ; #1扫码NG推料气缸缩回位
LD H73.13  ; #1扫码NG推料气缸伸出位屏蔽
AND 13.10  ; #1扫码NG推料气缸
ORLD
ANDLD
TIMX(550) 0261 D1561  ; #1扫码NG推料气缸伸出位屏蔽延时, #1扫码NG推料气缸伸出位
LD TR0
LD 7.00  ; #2扫码NG推料气缸缩回位
ANDNOT 7.01  ; #2扫码NG推料气缸伸出位
LD H73.14  ; #2扫码NG推料气缸缩回位屏蔽
ANDNOT 13.11  ; #2扫码NG推料气缸
ORLD
ANDLD
TIMX(550) 0262 D1562  ; #2扫码NG推料气缸缩回位屏蔽延时, #2扫码NG推料气缸缩回位
LD TR0
LD 7.01  ; #2扫码NG推料气缸伸出位
ANDNOT 7.00  ; #2扫码NG推料气缸缩回位
LD H73.15  ; #2扫码NG推料气缸伸出位屏蔽
AND 13.11  ; #2扫码NG推料气缸
ORLD
ANDLD
TIMX(550) 0263 D1563  ; #2扫码NG推料气缸伸出位屏蔽延时, #2扫码NG推料气缸伸出位
LD TR0
LD 7.02  ; #1测试NG推料气缸缩回位
ANDNOT 7.03  ; #1测试NG推料气缸伸出位
LD H74.00  ; #1测试NG推料气缸缩回位屏蔽
ANDNOT 13.12  ; #1测试NG推料气缸
ORLD
ANDLD
TIMX(550) 0264 D1564  ; #1测试NG推料气缸缩回位屏蔽延时, #1测试NG推料气缸缩回位
LD TR0
LD 7.03  ; #1测试NG推料气缸伸出位
ANDNOT 7.02  ; #1测试NG推料气缸缩回位
LD H74.01  ; #1测试NG推料气缸伸出位屏蔽
AND 13.12  ; #1测试NG推料气缸
ORLD
ANDLD
TIMX(550) 0265 D1565  ; #1测试NG推料气缸伸出屏蔽延时, #1测试NG推料气缸伸出延时
LD TR0
LD 7.04  ; #2测试NG推料气缸缩回位
ANDNOT 7.05  ; #2测试NG推料气缸伸出位
LD H74.02  ; #2测试NG推料气缸缩回位屏蔽
ANDNOT 13.13  ; #2测试NG推料气缸
ORLD
ANDLD
TIMX(550) 0266 D1566  ; #2测试NG推料气缸缩回位屏蔽延时, #2测试NG推料气缸缩回位
LD TR0
LD 7.05  ; #2测试NG推料气缸伸出位
ANDNOT 7.04  ; #2测试NG推料气缸缩回位
LD H74.03  ; #2测试NG推料气缸伸出位屏蔽
AND 13.13  ; #2测试NG推料气缸
ORLD
ANDLD
TIMX(550) 0267 D1567  ; #2测试NG推料气缸伸出位屏蔽延时, #2测试NG推料气缸伸出位

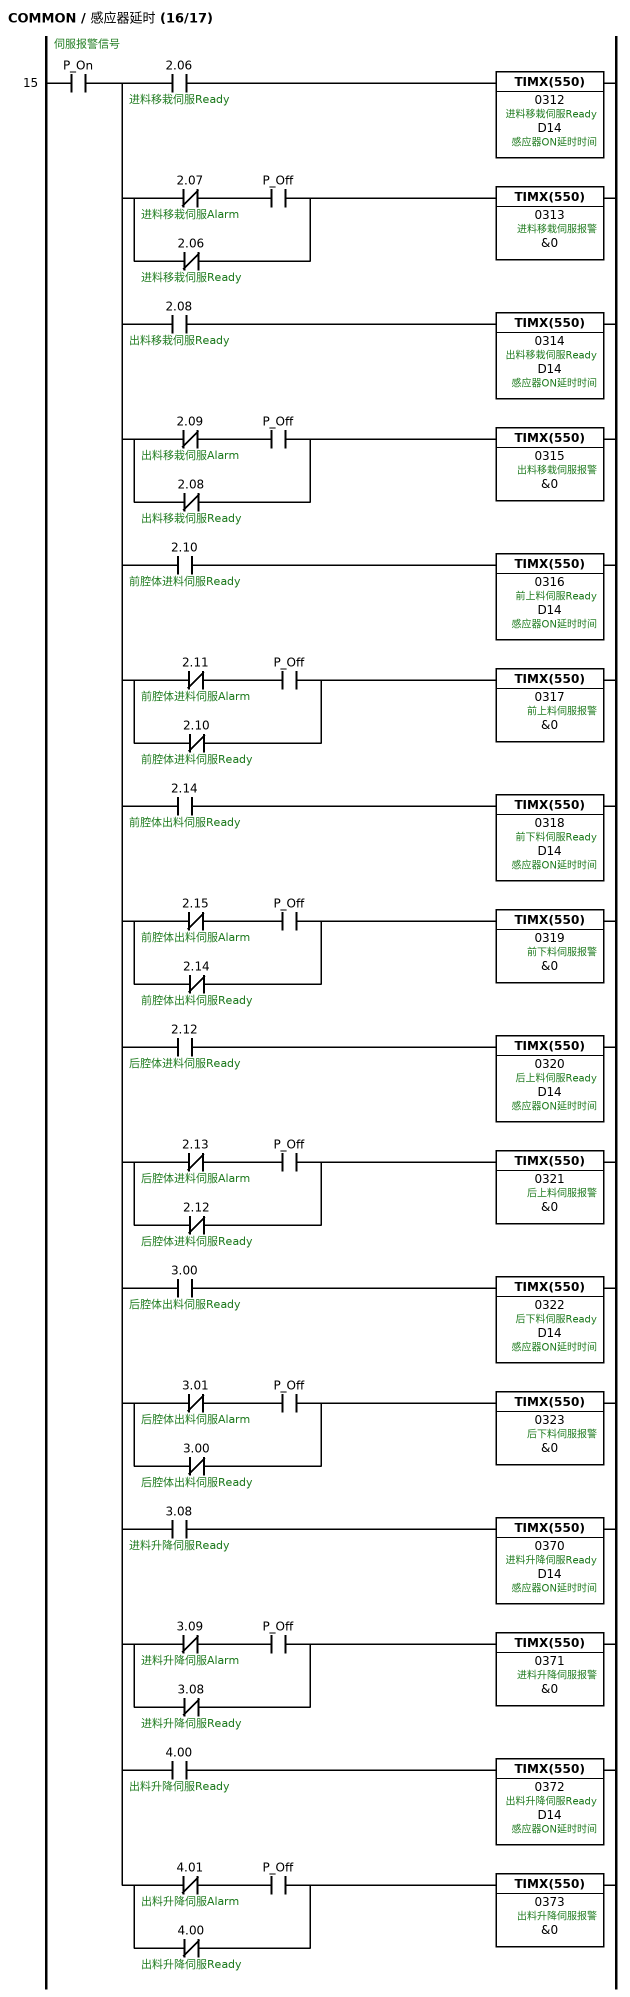
; rung 15: 伺服报警信号
LD P_On
OUT TR0
AND 2.06  ; 进料移栽伺服Ready
TIMX(550) 0312 D14  ; 感应器ON延时时间, 进料移栽伺服Ready
LD TR0
LDNOT 2.07  ; 进料移栽伺服Alarm
AND P_Off
ORNOT 2.06  ; 进料移栽伺服Ready
ANDLD
TIMX(550) 0313 &0  ; 进料移栽伺服报警
LD TR0
AND 2.08  ; 出料移栽伺服Ready
TIMX(550) 0314 D14  ; 感应器ON延时时间, 出料移栽伺服Ready
LD TR0
LDNOT 2.09  ; 出料移栽伺服Alarm
AND P_Off
ORNOT 2.08  ; 出料移栽伺服Ready
ANDLD
TIMX(550) 0315 &0  ; 出料移栽伺服报警
LD TR0
AND 2.10  ; 前腔体进料伺服Ready
TIMX(550) 0316 D14  ; 感应器ON延时时间, 前上料伺服Ready
LD TR0
LDNOT 2.11  ; 前腔体进料伺服Alarm
AND P_Off
ORNOT 2.10  ; 前腔体进料伺服Ready
ANDLD
TIMX(550) 0317 &0  ; 前上料伺服报警
LD TR0
AND 2.14  ; 前腔体出料伺服Ready
TIMX(550) 0318 D14  ; 感应器ON延时时间, 前下料伺服Ready
LD TR0
LDNOT 2.15  ; 前腔体出料伺服Alarm
AND P_Off
ORNOT 2.14  ; 前腔体出料伺服Ready
ANDLD
TIMX(550) 0319 &0  ; 前下料伺服报警
LD TR0
AND 2.12  ; 后腔体进料伺服Ready
TIMX(550) 0320 D14  ; 感应器ON延时时间, 后上料伺服Ready
LD TR0
LDNOT 2.13  ; 后腔体进料伺服Alarm
AND P_Off
ORNOT 2.12  ; 后腔体进料伺服Ready
ANDLD
TIMX(550) 0321 &0  ; 后上料伺服报警
LD TR0
AND 3.00  ; 后腔体出料伺服Ready
TIMX(550) 0322 D14  ; 感应器ON延时时间, 后下料伺服Ready
LD TR0
LDNOT 3.01  ; 后腔体出料伺服Alarm
AND P_Off
ORNOT 3.00  ; 后腔体出料伺服Ready
ANDLD
TIMX(550) 0323 &0  ; 后下料伺服报警
LD TR0
AND 3.08  ; 进料升降伺服Ready
TIMX(550) 0370 D14  ; 感应器ON延时时间, 进料升降伺服Ready
LD TR0
LDNOT 3.09  ; 进料升降伺服Alarm
AND P_Off
ORNOT 3.08  ; 进料升降伺服Ready
ANDLD
TIMX(550) 0371 &0  ; 进料升降伺服报警
LD TR0
AND 4.00  ; 出料升降伺服Ready
TIMX(550) 0372 D14  ; 感应器ON延时时间, 出料升降伺服Ready
LD TR0
LDNOT 4.01  ; 出料升降伺服Alarm
AND P_Off
ORNOT 4.00  ; 出料升降伺服Ready
ANDLD
TIMX(550) 0373 &0  ; 出料升降伺服报警

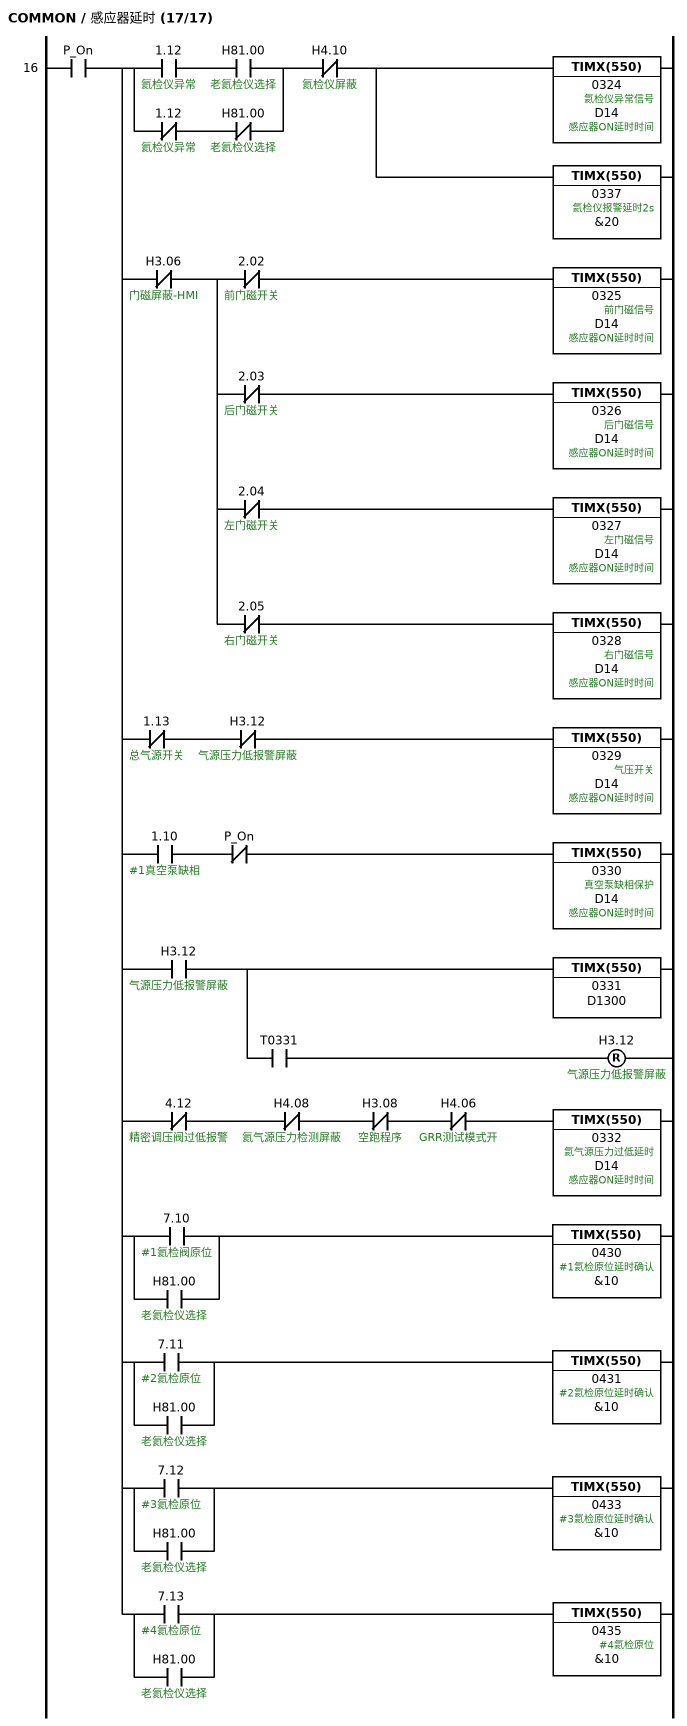
; rung 16
LD P_On
OUT TR0
LD 1.12  ; 氦检仪异常
AND H81.00  ; 老氦检仪选择
LDNOT 1.12  ; 氦检仪异常
ANDNOT H81.00  ; 老氦检仪选择
ORLD
ANDLD
ANDNOT H4.10  ; 氦检仪屏蔽
TIMX(550) 0324 D14  ; 感应器ON延时时间, 氦检仪异常信号
TIMX(550) 0337 &20  ; 氦检仪报警延时2s
LD TR0
ANDNOT H3.06  ; 门磁屏蔽-HMI
OUT TR1
ANDNOT 2.02  ; 前门磁开关
TIMX(550) 0325 D14  ; 感应器ON延时时间, 前门磁信号
LD TR1
ANDNOT 2.03  ; 后门磁开关
TIMX(550) 0326 D14  ; 感应器ON延时时间, 后门磁信号
LD TR1
ANDNOT 2.04  ; 左门磁开关
TIMX(550) 0327 D14  ; 感应器ON延时时间, 左门磁信号
LD TR1
ANDNOT 2.05  ; 右门磁开关
TIMX(550) 0328 D14  ; 感应器ON延时时间, 右门磁信号
LD TR0
ANDNOT 1.13  ; 总气源开关
ANDNOT H3.12  ; 气源压力低报警屏蔽
TIMX(550) 0329 D14  ; 感应器ON延时时间, 气压开关
LD TR0
AND 1.10  ; #1真空泵缺相
ANDNOT P_On
TIMX(550) 0330 D14  ; 感应器ON延时时间, 真空泵缺相保护
LD TR0
AND H3.12  ; 气源压力低报警屏蔽
TIMX(550) 0331 D1300
AND T0331
RSET H3.12  ; 气源压力低报警屏蔽
LD TR0
ANDNOT 4.12  ; 精密调压阀过低报警
ANDNOT H4.08  ; 氦气源压力检测屏蔽
ANDNOT H3.08  ; 空跑程序
ANDNOT H4.06  ; GRR测试模式开
TIMX(550) 0332 D14  ; 感应器ON延时时间, 氦气源压力过低延时
LD TR0
LD 7.10  ; #1氦检阀原位
OR H81.00  ; 老氦检仪选择
ANDLD
TIMX(550) 0430 &10  ; #1氦检原位延时确认
LD TR0
LD 7.11  ; #2氦检原位
OR H81.00  ; 老氦检仪选择
ANDLD
TIMX(550) 0431 &10  ; #2氦检原位延时确认
LD TR0
LD 7.12  ; #3氦检原位
OR H81.00  ; 老氦检仪选择
ANDLD
TIMX(550) 0433 &10  ; #3氦检原位延时确认
LD TR0
LD 7.13  ; #4氦检原位
OR H81.00  ; 老氦检仪选择
ANDLD
TIMX(550) 0435 &10  ; #4氦检原位

### Section 数据

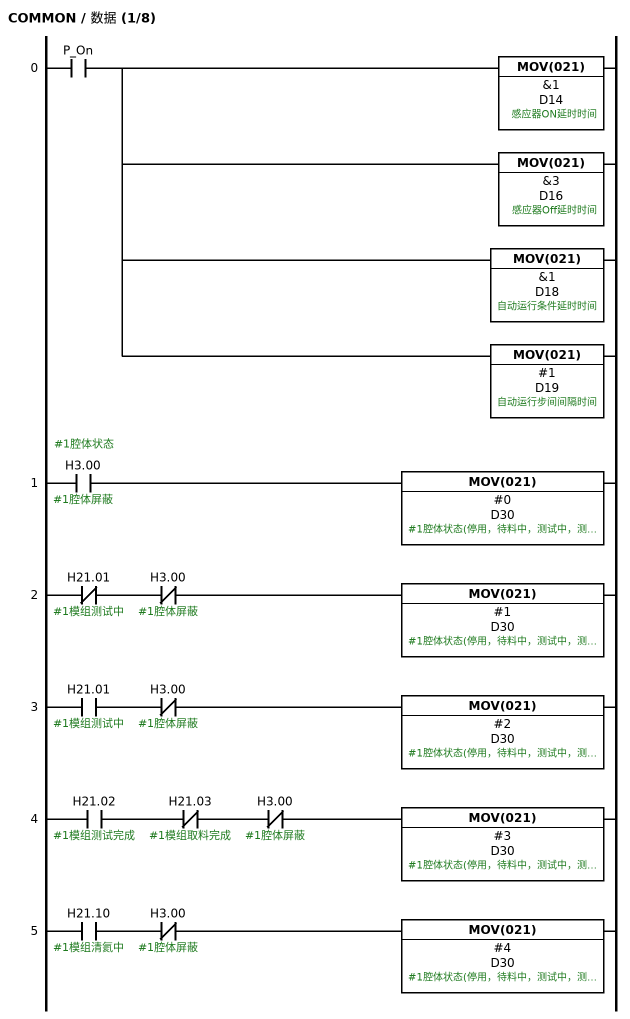
; rung 0
LD P_On
MOV(021) &1 D14  ; 感应器ON延时时间
MOV(021) &3 D16  ; 感应器Off延时时间
MOV(021) &1 D18  ; 自动运行条件延时时间
MOV(021) #1 D19  ; 自动运行步间间隔时间
; rung 1: #1腔体状态
LD H3.00  ; #1腔体屏蔽
MOV(021) #0 D30  ; #1腔体状态(停用，待料中，测试中，测试完成
; rung 2
LDNOT H21.01  ; #1模组测试中
ANDNOT H3.00  ; #1腔体屏蔽
MOV(021) #1 D30  ; #1腔体状态(停用，待料中，测试中，测试完成
; rung 3
LD H21.01  ; #1模组测试中
ANDNOT H3.00  ; #1腔体屏蔽
MOV(021) #2 D30  ; #1腔体状态(停用，待料中，测试中，测试完成
; rung 4
LD H21.02  ; #1模组测试完成
ANDNOT H21.03  ; #1模组取料完成
ANDNOT H3.00  ; #1腔体屏蔽
MOV(021) #3 D30  ; #1腔体状态(停用，待料中，测试中，测试完成
; rung 5
LD H21.10  ; #1模组清氦中
ANDNOT H3.00  ; #1腔体屏蔽
MOV(021) #4 D30  ; #1腔体状态(停用，待料中，测试中，测试完成

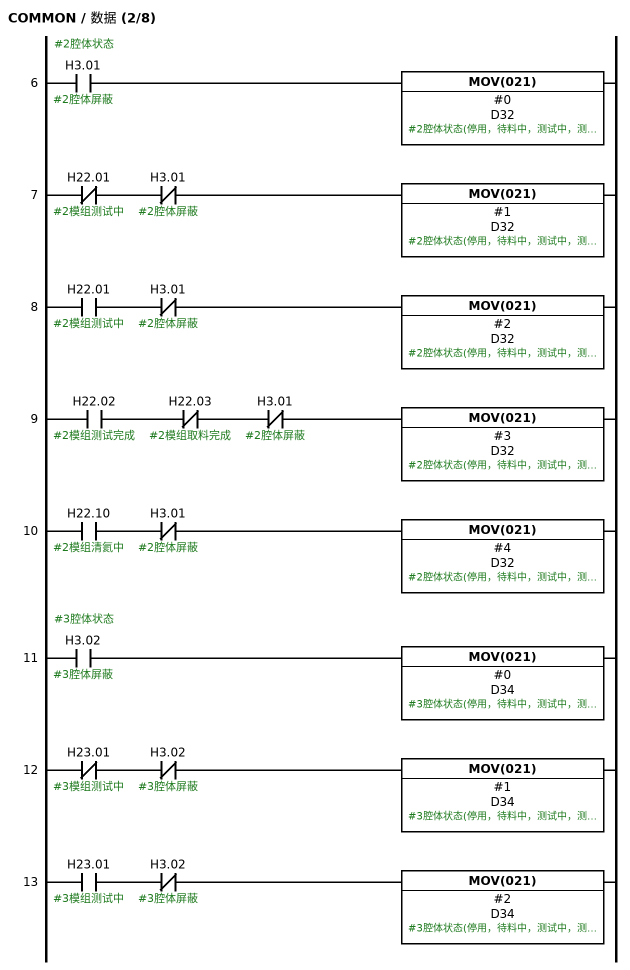
; rung 6: #2腔体状态
LD H3.01  ; #2腔体屏蔽
MOV(021) #0 D32  ; #2腔体状态(停用，待料中，测试中，测试完成
; rung 7
LDNOT H22.01  ; #2模组测试中
ANDNOT H3.01  ; #2腔体屏蔽
MOV(021) #1 D32  ; #2腔体状态(停用，待料中，测试中，测试完成
; rung 8
LD H22.01  ; #2模组测试中
ANDNOT H3.01  ; #2腔体屏蔽
MOV(021) #2 D32  ; #2腔体状态(停用，待料中，测试中，测试完成
; rung 9
LD H22.02  ; #2模组测试完成
ANDNOT H22.03  ; #2模组取料完成
ANDNOT H3.01  ; #2腔体屏蔽
MOV(021) #3 D32  ; #2腔体状态(停用，待料中，测试中，测试完成
; rung 10
LD H22.10  ; #2模组清氦中
ANDNOT H3.01  ; #2腔体屏蔽
MOV(021) #4 D32  ; #2腔体状态(停用，待料中，测试中，测试完成
; rung 11: #3腔体状态
LD H3.02  ; #3腔体屏蔽
MOV(021) #0 D34  ; #3腔体状态(停用，待料中，测试中，测试完成
; rung 12
LDNOT H23.01  ; #3模组测试中
ANDNOT H3.02  ; #3腔体屏蔽
MOV(021) #1 D34  ; #3腔体状态(停用，待料中，测试中，测试完成
; rung 13
LD H23.01  ; #3模组测试中
ANDNOT H3.02  ; #3腔体屏蔽
MOV(021) #2 D34  ; #3腔体状态(停用，待料中，测试中，测试完成

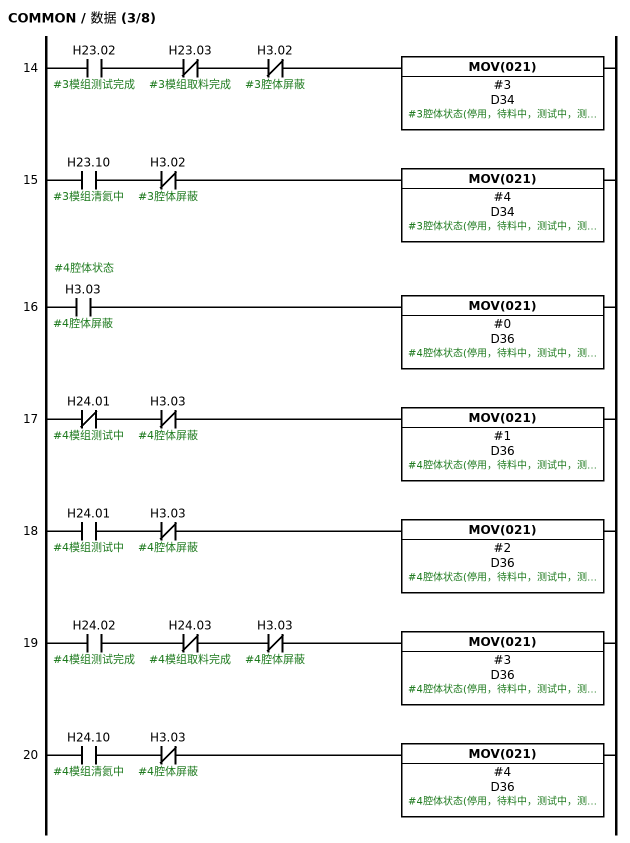
; rung 14
LD H23.02  ; #3模组测试完成
ANDNOT H23.03  ; #3模组取料完成
ANDNOT H3.02  ; #3腔体屏蔽
MOV(021) #3 D34  ; #3腔体状态(停用，待料中，测试中，测试完成
; rung 15
LD H23.10  ; #3模组清氦中
ANDNOT H3.02  ; #3腔体屏蔽
MOV(021) #4 D34  ; #3腔体状态(停用，待料中，测试中，测试完成
; rung 16: #4腔体状态
LD H3.03  ; #4腔体屏蔽
MOV(021) #0 D36  ; #4腔体状态(停用，待料中，测试中，测试完成
; rung 17
LDNOT H24.01  ; #4模组测试中
ANDNOT H3.03  ; #4腔体屏蔽
MOV(021) #1 D36  ; #4腔体状态(停用，待料中，测试中，测试完成
; rung 18
LD H24.01  ; #4模组测试中
ANDNOT H3.03  ; #4腔体屏蔽
MOV(021) #2 D36  ; #4腔体状态(停用，待料中，测试中，测试完成
; rung 19
LD H24.02  ; #4模组测试完成
ANDNOT H24.03  ; #4模组取料完成
ANDNOT H3.03  ; #4腔体屏蔽
MOV(021) #3 D36  ; #4腔体状态(停用，待料中，测试中，测试完成
; rung 20
LD H24.10  ; #4模组清氦中
ANDNOT H3.03  ; #4腔体屏蔽
MOV(021) #4 D36  ; #4腔体状态(停用，待料中，测试中，测试完成

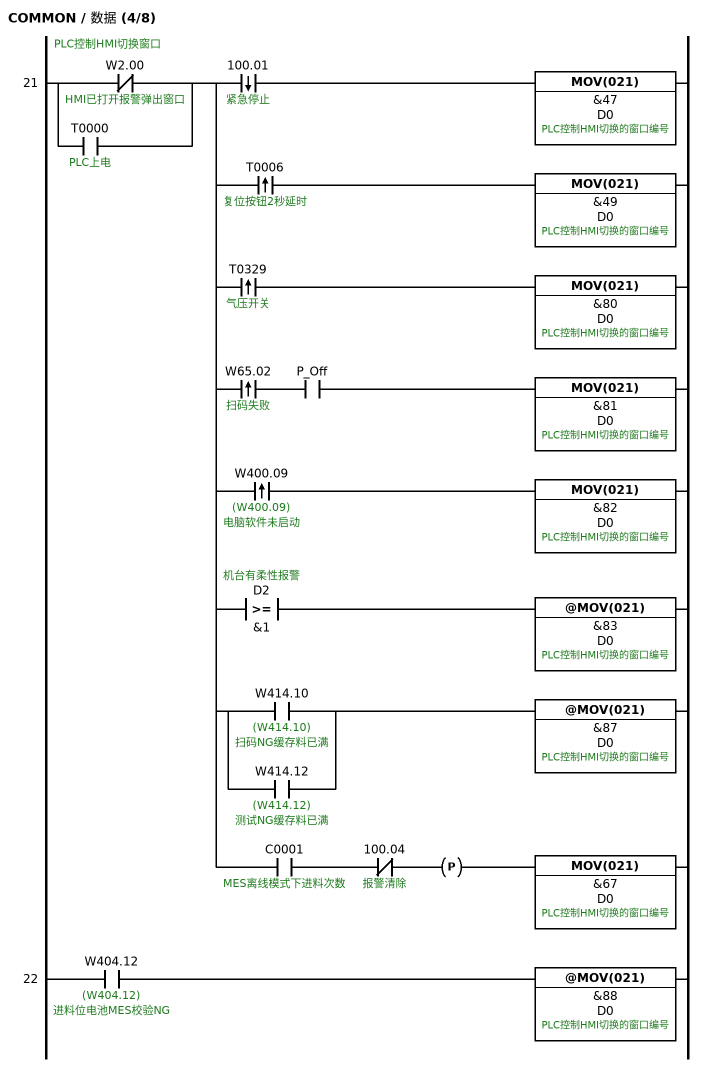
; rung 21: PLC控制HMI切换窗口
LDNOT W2.00  ; HMI已打开报警弹出窗口
OR T0000  ; PLC上电
OUT TR0
%AND 100.01  ; 紧急停止
MOV(021) &47 D0  ; PLC控制HMI切换的窗口编号
LD TR0
@AND T0006  ; 复位按钮2秒延时
MOV(021) &49 D0  ; PLC控制HMI切换的窗口编号
LD TR0
@AND T0329  ; 气压开关
MOV(021) &80 D0  ; PLC控制HMI切换的窗口编号
LD TR0
@AND W65.02  ; 扫码失败
AND P_Off
MOV(021) &81 D0  ; PLC控制HMI切换的窗口编号
LD TR0
@AND W400.09  ; (W400.09) 电脑软件未启动
MOV(021) &82 D0  ; PLC控制HMI切换的窗口编号
LD TR0
AND>=(325) D2 &1  ; 机台有柔性报警
@MOV(021) &83 D0  ; PLC控制HMI切换的窗口编号
LD TR0
LD W414.10  ; (W414.10) 扫码NG缓存料已满
OR W414.12  ; (W414.12) 测试NG缓存料已满
ANDLD
@MOV(021) &87 D0  ; PLC控制HMI切换的窗口编号
LD TR0
AND C0001  ; MES离线模式下进料次数
ANDNOT 100.04  ; 报警清除
UP(521)
MOV(021) &67 D0  ; PLC控制HMI切换的窗口编号
; rung 22
LD W404.12  ; (W404.12) 进料位电池MES校验NG
@MOV(021) &88 D0  ; PLC控制HMI切换的窗口编号

